SPLINE
SPL {X  -158.264, Y  +691.203, Z    +0.000, E1   -17.264, E3 +51603.968}
SPL {X  -159.000, Y  +685.560, Z    +0.000, E1   -12.398, E3 +51625.143}
SPL {X  -159.924, Y  +672.625, Z    +0.000, E1    -3.689, E3 +51640.160}
SPL {X  -160.000, Y  +663.203, Z    +0.000, E1    +3.155, E3 +51646.815}
SPL {X  -160.000, Y  +652.103, Z    +0.000, E1   +11.247, E3 +51658.485}
SPL {X  -160.000, Y  +641.822, Z    +0.000, E1   +17.059, E3 +51677.859}
SPL {X  -160.000, Y  +631.293, Z    +0.000, E1   +20.354, E3 +51711.738}
SPL {X  -160.000, Y  +627.542, Z    +0.000, E1   +20.380, E3 +51733.145}
SPL {X  -160.000, Y  +623.532, Z    +0.000, E1   +20.378, E3 +51756.111}
SPL {X  -160.000, Y  +619.329, Z    +0.000, E1   +20.391, E3 +51780.148}
SPL {X  -160.000, Y  +614.967, Z    +0.000, E1   +20.392, E3 +51805.128}
SPL {X  -160.000, Y  +611.206, Z    +0.000, E1   +20.351, E3 +51826.800}
SPL {X  -160.000, Y  +607.824, Z    +0.000, E1   +20.354, E3 +51846.221}
SPL {X  -160.000, Y  +603.899, Z    +0.000, E1   +20.373, E3 +51868.671}
SPL {X  -160.000, Y  +599.617, Z    +0.000, E1   +20.384, E3 +51893.164}
SPL {X  -160.000, Y  +595.532, Z    +0.000, E1   +20.373, E3 +51916.525}
SPL {X  -160.000, Y  +591.705, Z    +0.000, E1   +20.373, E3 +51938.450}
SPL {X  -160.000, Y  +588.037, Z    +0.000, E1   +20.359, E3 +51959.537}
SPL {X  -160.000, Y  +584.320, Z    +0.000, E1   +20.364, E3 +51980.838}
SPL {X  -160.000, Y  +580.616, Z    +0.000, E1   +20.357, E3 +52002.065}
SPL {X  -160.000, Y  +577.083, Z    +0.000, E1   +20.358, E3 +52022.314}
SPL {X  -160.000, Y  +573.158, Z    +0.000, E1   +20.377, E3 +52044.766}
SPL {X  -160.000, Y  +568.802, Z    +0.000, E1   +20.385, E3 +52069.718}
SPL {X  -160.000, Y  +564.937, Z    +0.000, E1   +20.350, E3 +52091.938}
SPL {X  -160.000, Y  +561.213, Z    +0.000, E1   +20.372, E3 +52113.225}
SPL {X  -160.000, Y  +557.320, Z    +0.000, E1   +20.363, E3 +52135.551}
SPL {X  -160.000, Y  +553.712, Z    +0.000, E1   +20.355, E3 +52156.251}
SPL {X  -160.000, Y  +550.040, Z    +0.000, E1   +20.360, E3 +52177.289}
SPL {X  -160.000, Y  +546.180, Z    +0.000, E1   +20.370, E3 +52199.345}
SPL {X  -160.000, Y  +542.032, Z    +0.000, E1   +20.384, E3 +52223.084}
SPL {X  -160.000, Y  +537.870, Z    +0.000, E1   +20.372, E3 +52246.959}
SPL {X  -160.000, Y  +534.086, Z    +0.000, E1   +20.356, E3 +52268.713}
SPL {X  -160.000, Y  +530.164, Z    +0.000, E1   +20.382, E3 +52291.063}
SPL {X  -160.000, Y  +527.505, Z    +0.000, E1   +20.318, E3 +52306.436}
SPL {X  -160.000, Y  +511.620, Z    +0.000, E1   +28.365, E3 +52316.899}
SPL {X  -160.000, Y  +507.906, Z    +0.000, E1   +28.152, E3 +52333.295}
SPL {X  -160.000, Y  +506.085, Z    +0.000, E1   +26.146, E3 +52355.754}
SPL {X  -160.000, Y  +504.342, Z    +0.000, E1   +24.109, E3 +52379.269}
SPL {X  -160.000, Y  +503.002, Z    +0.000, E1   +22.325, E3 +52400.275}
SPL {X  -160.000, Y  +500.783, Z    +0.000, E1   +21.421, E3 +52419.864}
SPL {X  -160.000, Y  +497.229, Z    +0.000, E1   +21.403, E3 +52439.172}
SPL {X  -160.000, Y  +493.901, Z    +0.000, E1   +21.409, E3 +52457.191}
SPL {X  -160.000, Y  +490.791, Z    +0.000, E1   +21.400, E3 +52474.064}
SPL {X  -160.000, Y  +487.647, Z    +0.000, E1   +21.401, E3 +52491.110}
SPL {X  -160.000, Y  +484.273, Z    +0.000, E1   +21.408, E3 +52509.390}
SPL {X  -160.000, Y  +481.093, Z    +0.000, E1   +21.389, E3 +52526.699}
SPL {X  -160.000, Y  +478.021, Z    +0.000, E1   +21.401, E3 +52543.306}
SPL {X  -160.000, Y  +474.639, Z    +0.000, E1   +21.410, E3 +52561.597}
SPL {X  -160.000, Y  +471.343, Z    +0.000, E1   +21.399, E3 +52579.499}
SPL {X  -160.000, Y  +468.133, Z    +0.000, E1   +21.402, E3 +52596.891}
SPL {X  -160.000, Y  +464.638, Z    +0.000, E1   +21.421, E3 +52615.740}
SPL {X  -160.000, Y  +461.045, Z    +0.000, E1   +21.424, E3 +52635.154}
SPL {X  -160.000, Y  +457.606, Z    +0.000, E1   +21.413, E3 +52653.864}
SPL {X  -160.000, Y  +454.417, Z    +0.000, E1   +21.401, E3 +52671.172}
SPL {X  -160.000, Y  +451.425, Z    +0.000, E1   +21.404, E3 +52687.394}
SPL {X  -160.000, Y  +448.039, Z    +0.000, E1   +21.417, E3 +52705.687}
SPL {X  -160.000, Y  +444.787, Z    +0.000, E1   +21.414, E3 +52723.242}
SPL {X  -160.000, Y  +441.637, Z    +0.000, E1   +21.431, E3 +52740.220}
SPL {X  -160.000, Y  +438.199, Z    +0.000, E1   +21.432, E3 +52758.824}
SPL {X  -160.000, Y  +434.875, Z    +0.000, E1   +21.424, E3 +52776.864}
SPL {X  -160.000, Y  +431.689, Z    +0.000, E1   +21.423, E3 +52794.112}
SPL {X  -160.000, Y  +428.451, Z    +0.000, E1   +21.430, E3 +52811.592}
SPL {X  -160.000, Y  +425.120, Z    +0.000, E1   +21.430, E3 +52829.656}
SPL {X  -160.000, Y  +421.671, Z    +0.000, E1   +21.430, E3 +52848.340}
SPL {X  -160.000, Y  +418.225, Z    +0.000, E1   +21.425, E3 +52867.021}
SPL {X  -160.000, Y  +414.956, Z    +0.000, E1   +21.424, E3 +52884.702}
SPL {X  -160.000, Y  +411.834, Z    +0.000, E1   +21.420, E3 +52901.620}
SPL {X  -160.000, Y  +408.570, Z    +0.000, E1   +21.432, E3 +52919.229}
SPL {X  -160.000, Y  +405.237, Z    +0.000, E1   +21.432, E3 +52937.258}
SPL {X  -160.000, Y  +402.004, Z    +0.000, E1   +21.424, E3 +52954.833}
SPL {X  -160.000, Y  +398.626, Z    +0.000, E1   +21.425, E3 +52973.139}
SPL {X  -160.000, Y  +395.405, Z    +0.000, E1   +21.422, E3 +52990.557}
SPL {X  -160.000, Y  +392.641, Z    +0.000, E1   +21.407, E3 +53005.555}
SPL {X  -159.989, Y  +390.129, Z    +0.000, E1   +21.406, E3 +53019.196}
SPL {X  -159.932, Y  +387.337, Z    +0.000, E1   +21.403, E3 +53034.392}
SPL {X  -159.823, Y  +384.478, Z    +0.000, E1   +21.379, E3 +53050.055}
SPL {X  -159.660, Y  +381.581, Z    +0.000, E1   +21.363, E3 +53065.943}
SPL {X  -159.452, Y  +378.773, Z    +0.000, E1   +21.330, E3 +53081.390}
SPL {X  -159.222, Y  +376.244, Z    +0.000, E1   +21.297, E3 +53095.352}
SPL {X  -158.814, Y  +372.556, Z    +0.000, E1   +21.316, E3 +53115.619}
SPL {X  -158.301, Y  +368.743, Z    +0.000, E1   +21.199, E3 +53136.941}
SPL {X  -157.981, Y  +366.660, Z    +0.000, E1   +19.986, E3 +53159.909}
ENDSPLINE

SPLINE
SPL {X  -158.491, Y  +370.077, Z    +0.000, E1   +15.910, E3 +53184.922}
SPL {X  -159.771, Y  +383.450, Z    +0.000, E1    +6.314, E3 +53208.077}
SPL {X  -160.000, Y  +392.463, Z    +0.000, E1    +0.112, E3 +53214.584}
SPL {X  -160.000, Y  +399.874, Z    +0.000, E1    -5.508, E3 +53219.086}
SPL {X  -160.000, Y  +411.622, Z    +0.000, E1   -13.815, E3 +53231.206}
SPL {X  -160.000, Y  +419.836, Z    +0.000, E1   -18.198, E3 +53246.380}
SPL {X  -160.000, Y  +430.523, Z    +0.000, E1   -21.710, E3 +53276.580}
SPL {X  -160.000, Y  +433.426, Z    +0.000, E1   -21.735, E3 +53291.994}
SPL {X  -160.000, Y  +436.131, Z    +0.000, E1   -21.710, E3 +53306.469}
SPL {X  -160.000, Y  +439.046, Z    +0.000, E1   -21.732, E3 +53321.963}
SPL {X  -160.000, Y  +442.009, Z    +0.000, E1   -21.719, E3 +53337.785}
SPL {X  -160.000, Y  +444.891, Z    +0.000, E1   -21.724, E3 +53353.140}
SPL {X  -160.000, Y  +449.017, Z    +0.000, E1   -21.792, E3 +53374.932}
SPL {X  -160.000, Y  +452.864, Z    +0.000, E1   -21.730, E3 +53395.550}
SPL {X  -160.000, Y  +455.470, Z    +0.000, E1   -21.722, E3 +53409.439}
SPL {X  -160.000, Y  +458.295, Z    +0.000, E1   -21.738, E3 +53424.460}
SPL {X  -160.000, Y  +461.133, Z    +0.000, E1   -21.720, E3 +53439.642}
SPL {X  -160.000, Y  +464.458, Z    +0.000, E1   -21.770, E3 +53457.161}
SPL {X  -160.000, Y  +468.250, Z    +0.000, E1   -21.764, E3 +53477.314}
SPL {X  -160.000, Y  +472.226, Z    +0.000, E1   -21.782, E3 +53498.473}
SPL {X  -160.000, Y  +476.333, Z    +0.000, E1   -21.767, E3 +53520.387}
SPL {X  -160.000, Y  +480.244, Z    +0.000, E1   -21.765, E3 +53541.252}
SPL {X  -160.000, Y  +484.301, Z    +0.000, E1   -21.775, E3 +53562.780}
SPL {X  -160.000, Y  +488.201, Z    +0.000, E1   -21.768, E3 +53583.540}
SPL {X  -160.000, Y  +492.394, Z    +0.000, E1   -21.802, E3 +53605.714}
SPL {X  -160.000, Y  +496.781, Z    +0.000, E1   -21.798, E3 +53629.026}
SPL {X  -160.000, Y  +501.083, Z    +0.000, E1   -21.796, E3 +53651.956}
SPL {X  -160.000, Y  +504.917, Z    +0.000, E1   -21.764, E3 +53672.460}
SPL {X  -160.000, Y  +508.886, Z    +0.000, E1   -21.791, E3 +53693.546}
SPL {X  -160.000, Y  +513.057, Z    +0.000, E1   -21.767, E3 +53715.854}
SPL {X  -160.000, Y  +517.221, Z    +0.000, E1   -21.778, E3 +53738.006}
SPL {X  -160.000, Y  +521.677, Z    +0.000, E1   -21.781, E3 +53761.768}
SPL {X  -160.000, Y  +525.729, Z    +0.000, E1   -21.753, E3 +53783.407}
SPL {X  -160.000, Y  +529.456, Z    +0.000, E1   -21.766, E3 +53803.186}
SPL {X  -160.000, Y  +533.608, Z    +0.000, E1   -21.776, E3 +53825.317}
SPL {X  -160.000, Y  +538.227, Z    +0.000, E1   -21.794, E3 +53849.849}
SPL {X  -160.000, Y  +542.483, Z    +0.000, E1   -21.764, E3 +53872.574}
SPL {X  -160.000, Y  +546.194, Z    +0.000, E1   -21.754, E3 +53892.391}
SPL {X  -160.000, Y  +550.131, Z    +0.000, E1   -21.771, E3 +53913.327}
SPL {X  -160.000, Y  +554.462, Z    +0.000, E1   -21.777, E3 +53936.381}
SPL {X  -160.000, Y  +558.542, Z    +0.000, E1   -21.758, E3 +53958.153}
SPL {X  -160.000, Y  +562.615, Z    +0.000, E1   -21.776, E3 +53979.809}
SPL {X  -160.000, Y  +566.764, Z    +0.000, E1   -21.764, E3 +54001.934}
SPL {X  -160.000, Y  +570.657, Z    +0.000, E1   -21.758, E3 +54022.681}
SPL {X  -160.000, Y  +574.688, Z    +0.000, E1   -21.771, E3 +54044.124}
SPL {X  -160.000, Y  +578.864, Z    +0.000, E1   -21.770, E3 +54066.375}
SPL {X  -160.000, Y  +582.807, Z    +0.000, E1   -21.754, E3 +54087.429}
SPL {X  -160.000, Y  +586.993, Z    +0.000, E1   -21.779, E3 +54109.665}
SPL {X  -160.000, Y  +591.368, Z    +0.000, E1   -21.775, E3 +54132.952}
SPL {X  -160.000, Y  +595.703, Z    +0.000, E1   -21.775, E3 +54156.061}
SPL {X  -160.000, Y  +599.558, Z    +0.000, E1   -21.748, E3 +54176.639}
SPL {X  -160.000, Y  +603.126, Z    +0.000, E1   -21.757, E3 +54195.618}
SPL {X  -160.000, Y  +607.107, Z    +0.000, E1   -21.766, E3 +54216.843}
SPL {X  -160.000, Y  +611.246, Z    +0.000, E1   -21.760, E3 +54238.917}
SPL {X  -160.000, Y  +615.151, Z    +0.000, E1   -21.752, E3 +54259.730}
SPL {X  -160.000, Y  +618.728, Z    +0.000, E1   -21.747, E3 +54278.792}
SPL {X  -160.000, Y  +622.318, Z    +0.000, E1   -21.753, E3 +54297.907}
SPL {X  -160.000, Y  +625.877, Z    +0.000, E1   -21.745, E3 +54316.885}
SPL {X  -160.000, Y  +629.892, Z    +0.000, E1   -21.777, E3 +54338.209}
SPL {X  -160.000, Y  +634.024, Z    +0.000, E1   -21.756, E3 +54360.259}
SPL {X  -160.000, Y  +637.661, Z    +0.000, E1   -21.748, E3 +54379.650}
SPL {X  -160.000, Y  +641.244, Z    +0.000, E1   -21.752, E3 +54398.721}
SPL {X  -160.000, Y  +645.120, Z    +0.000, E1   -21.762, E3 +54419.353}
SPL {X  -160.000, Y  +649.214, Z    +0.000, E1   -21.766, E3 +54441.141}
SPL {X  -160.000, Y  +653.188, Z    +0.000, E1   -21.771, E3 +54462.204}
SPL {X  -160.000, Y  +656.905, Z    +0.000, E1   -21.769, E3 +54481.979}
SPL {X  -160.000, Y  +660.685, Z    +0.000, E1   -21.769, E3 +54502.147}
SPL {X  -160.000, Y  +664.985, Z    +0.000, E1   -21.790, E3 +54525.000}
SPL {X  -159.993, Y  +669.170, Z    +0.000, E1   -21.763, E3 +54547.358}
SPL {X  -159.916, Y  +672.869, Z    +0.000, E1   -21.755, E3 +54567.103}
SPL {X  -159.752, Y  +676.610, Z    +0.000, E1   -21.740, E3 +54587.178}
SPL {X  -159.478, Y  +680.618, Z    +0.000, E1   -21.719, E3 +54608.777}
SPL {X  -159.108, Y  +684.576, Z    +0.000, E1   -21.664, E3 +54630.247}
SPL {X  -158.638, Y  +688.530, Z    +0.000, E1   -21.617, E3 +54651.768}
SPL {X  -158.097, Y  +692.303, Z    +0.000, E1   -21.529, E3 +54672.486}
ENDSPLINE

SPLINE
SPL {X  -158.264, Y  +691.203, Z    +0.000, E1   -17.264, E3 +54709.231}
SPL {X  -159.000, Y  +685.560, Z    +0.000, E1   -12.398, E3 +54730.407}
SPL {X  -159.924, Y  +672.625, Z    +0.000, E1    -3.689, E3 +54745.424}
SPL {X  -160.000, Y  +663.203, Z    +0.000, E1    +3.155, E3 +54752.078}
SPL {X  -160.000, Y  +652.103, Z    +0.000, E1   +11.247, E3 +54763.748}
SPL {X  -160.000, Y  +641.822, Z    +0.000, E1   +17.059, E3 +54783.122}
SPL {X  -160.000, Y  +631.293, Z    +0.000, E1   +20.354, E3 +54817.002}
SPL {X  -160.000, Y  +627.542, Z    +0.000, E1   +20.380, E3 +54838.409}
SPL {X  -160.000, Y  +623.532, Z    +0.000, E1   +20.378, E3 +54861.374}
SPL {X  -160.000, Y  +619.329, Z    +0.000, E1   +20.391, E3 +54885.412}
SPL {X  -160.000, Y  +614.967, Z    +0.000, E1   +20.392, E3 +54910.392}
SPL {X  -160.000, Y  +611.206, Z    +0.000, E1   +20.351, E3 +54932.063}
SPL {X  -160.000, Y  +607.824, Z    +0.000, E1   +20.354, E3 +54951.484}
SPL {X  -160.000, Y  +603.899, Z    +0.000, E1   +20.373, E3 +54973.934}
SPL {X  -160.000, Y  +599.617, Z    +0.000, E1   +20.384, E3 +54998.428}
SPL {X  -160.000, Y  +595.532, Z    +0.000, E1   +20.373, E3 +55021.788}
SPL {X  -160.000, Y  +591.705, Z    +0.000, E1   +20.373, E3 +55043.713}
SPL {X  -160.000, Y  +588.037, Z    +0.000, E1   +20.359, E3 +55064.800}
SPL {X  -160.000, Y  +584.320, Z    +0.000, E1   +20.364, E3 +55086.102}
SPL {X  -160.000, Y  +580.616, Z    +0.000, E1   +20.357, E3 +55107.329}
SPL {X  -160.000, Y  +577.083, Z    +0.000, E1   +20.358, E3 +55127.577}
SPL {X  -160.000, Y  +573.158, Z    +0.000, E1   +20.377, E3 +55150.029}
SPL {X  -160.000, Y  +568.802, Z    +0.000, E1   +20.385, E3 +55174.981}
SPL {X  -160.000, Y  +564.937, Z    +0.000, E1   +20.350, E3 +55197.202}
SPL {X  -160.000, Y  +561.213, Z    +0.000, E1   +20.372, E3 +55218.488}
SPL {X  -160.000, Y  +557.320, Z    +0.000, E1   +20.363, E3 +55240.815}
SPL {X  -160.000, Y  +553.712, Z    +0.000, E1   +20.355, E3 +55261.514}
SPL {X  -160.000, Y  +550.040, Z    +0.000, E1   +20.360, E3 +55282.552}
SPL {X  -160.000, Y  +546.180, Z    +0.000, E1   +20.370, E3 +55304.608}
SPL {X  -160.000, Y  +542.032, Z    +0.000, E1   +20.384, E3 +55328.347}
SPL {X  -160.000, Y  +537.870, Z    +0.000, E1   +20.372, E3 +55352.223}
SPL {X  -160.000, Y  +534.086, Z    +0.000, E1   +20.356, E3 +55373.977}
SPL {X  -160.000, Y  +530.164, Z    +0.000, E1   +20.382, E3 +55396.326}
SPL {X  -160.000, Y  +527.505, Z    +0.000, E1   +20.318, E3 +55411.700}
SPL {X  -160.000, Y  +511.620, Z    +0.000, E1   +28.365, E3 +55422.163}
SPL {X  -160.000, Y  +507.906, Z    +0.000, E1   +28.152, E3 +55438.558}
SPL {X  -160.000, Y  +506.085, Z    +0.000, E1   +26.146, E3 +55461.018}
SPL {X  -160.000, Y  +504.342, Z    +0.000, E1   +24.109, E3 +55484.533}
SPL {X  -160.000, Y  +503.002, Z    +0.000, E1   +22.325, E3 +55505.538}
SPL {X  -160.000, Y  +500.783, Z    +0.000, E1   +21.421, E3 +55525.127}
SPL {X  -160.000, Y  +497.229, Z    +0.000, E1   +21.403, E3 +55544.435}
SPL {X  -160.000, Y  +493.901, Z    +0.000, E1   +21.409, E3 +55562.454}
SPL {X  -160.000, Y  +490.791, Z    +0.000, E1   +21.400, E3 +55579.327}
SPL {X  -160.000, Y  +487.647, Z    +0.000, E1   +21.401, E3 +55596.374}
SPL {X  -160.000, Y  +484.273, Z    +0.000, E1   +21.408, E3 +55614.654}
SPL {X  -160.000, Y  +481.093, Z    +0.000, E1   +21.389, E3 +55631.963}
SPL {X  -160.000, Y  +478.021, Z    +0.000, E1   +21.401, E3 +55648.569}
SPL {X  -160.000, Y  +474.639, Z    +0.000, E1   +21.410, E3 +55666.861}
SPL {X  -160.000, Y  +471.343, Z    +0.000, E1   +21.399, E3 +55684.763}
SPL {X  -160.000, Y  +468.133, Z    +0.000, E1   +21.402, E3 +55702.154}
SPL {X  -160.000, Y  +464.638, Z    +0.000, E1   +21.421, E3 +55721.003}
SPL {X  -160.000, Y  +461.045, Z    +0.000, E1   +21.424, E3 +55740.417}
SPL {X  -160.000, Y  +457.606, Z    +0.000, E1   +21.413, E3 +55759.127}
SPL {X  -160.000, Y  +454.417, Z    +0.000, E1   +21.401, E3 +55776.436}
SPL {X  -160.000, Y  +451.425, Z    +0.000, E1   +21.404, E3 +55792.657}
SPL {X  -160.000, Y  +448.039, Z    +0.000, E1   +21.417, E3 +55810.950}
SPL {X  -160.000, Y  +444.787, Z    +0.000, E1   +21.414, E3 +55828.505}
SPL {X  -160.000, Y  +441.637, Z    +0.000, E1   +21.431, E3 +55845.483}
SPL {X  -160.000, Y  +438.199, Z    +0.000, E1   +21.432, E3 +55864.087}
SPL {X  -160.000, Y  +434.875, Z    +0.000, E1   +21.424, E3 +55882.127}
SPL {X  -160.000, Y  +431.689, Z    +0.000, E1   +21.423, E3 +55899.375}
SPL {X  -160.000, Y  +428.451, Z    +0.000, E1   +21.430, E3 +55916.855}
SPL {X  -160.000, Y  +425.120, Z    +0.000, E1   +21.430, E3 +55934.919}
SPL {X  -160.000, Y  +421.671, Z    +0.000, E1   +21.430, E3 +55953.603}
SPL {X  -160.000, Y  +418.225, Z    +0.000, E1   +21.425, E3 +55972.285}
SPL {X  -160.000, Y  +414.956, Z    +0.000, E1   +21.424, E3 +55989.966}
SPL {X  -160.000, Y  +411.834, Z    +0.000, E1   +21.420, E3 +56006.884}
SPL {X  -160.000, Y  +408.570, Z    +0.000, E1   +21.432, E3 +56024.493}
SPL {X  -160.000, Y  +405.237, Z    +0.000, E1   +21.432, E3 +56042.521}
SPL {X  -160.000, Y  +402.004, Z    +0.000, E1   +21.424, E3 +56060.097}
SPL {X  -160.000, Y  +398.626, Z    +0.000, E1   +21.425, E3 +56078.403}
SPL {X  -160.000, Y  +395.405, Z    +0.000, E1   +21.422, E3 +56095.820}
SPL {X  -160.000, Y  +392.641, Z    +0.000, E1   +21.407, E3 +56110.819}
SPL {X  -159.989, Y  +390.129, Z    +0.000, E1   +21.406, E3 +56124.459}
SPL {X  -159.932, Y  +387.337, Z    +0.000, E1   +21.403, E3 +56139.655}
SPL {X  -159.823, Y  +384.478, Z    +0.000, E1   +21.379, E3 +56155.318}
SPL {X  -159.660, Y  +381.581, Z    +0.000, E1   +21.363, E3 +56171.207}
SPL {X  -159.452, Y  +378.773, Z    +0.000, E1   +21.330, E3 +56186.653}
SPL {X  -159.222, Y  +376.244, Z    +0.000, E1   +21.297, E3 +56200.615}
SPL {X  -158.814, Y  +372.556, Z    +0.000, E1   +21.316, E3 +56220.883}
SPL {X  -158.301, Y  +368.743, Z    +0.000, E1   +21.199, E3 +56242.205}
SPL {X  -157.981, Y  +366.660, Z    +0.000, E1   +19.986, E3 +56265.172}
ENDSPLINE

SPLINE
SPL {X  -158.491, Y  +370.077, Z    +0.000, E1   +15.910, E3 +56290.185}
SPL {X  -159.771, Y  +383.450, Z    +0.000, E1    +6.314, E3 +56313.340}
SPL {X  -160.000, Y  +392.463, Z    +0.000, E1    +0.112, E3 +56319.847}
SPL {X  -160.000, Y  +399.874, Z    +0.000, E1    -5.508, E3 +56324.350}
SPL {X  -160.000, Y  +411.622, Z    +0.000, E1   -13.815, E3 +56336.470}
SPL {X  -160.000, Y  +419.836, Z    +0.000, E1   -18.198, E3 +56351.643}
SPL {X  -160.000, Y  +430.523, Z    +0.000, E1   -21.710, E3 +56381.843}
SPL {X  -160.000, Y  +433.426, Z    +0.000, E1   -21.735, E3 +56397.258}
SPL {X  -160.000, Y  +436.131, Z    +0.000, E1   -21.710, E3 +56411.733}
SPL {X  -160.000, Y  +439.046, Z    +0.000, E1   -21.732, E3 +56427.226}
SPL {X  -160.000, Y  +442.009, Z    +0.000, E1   -21.719, E3 +56443.048}
SPL {X  -160.000, Y  +444.891, Z    +0.000, E1   -21.724, E3 +56458.404}
SPL {X  -160.000, Y  +449.017, Z    +0.000, E1   -21.792, E3 +56480.196}
SPL {X  -160.000, Y  +452.864, Z    +0.000, E1   -21.730, E3 +56500.813}
SPL {X  -160.000, Y  +455.470, Z    +0.000, E1   -21.722, E3 +56514.702}
SPL {X  -160.000, Y  +458.295, Z    +0.000, E1   -21.738, E3 +56529.723}
SPL {X  -160.000, Y  +461.133, Z    +0.000, E1   -21.720, E3 +56544.906}
SPL {X  -160.000, Y  +464.458, Z    +0.000, E1   -21.770, E3 +56562.425}
SPL {X  -160.000, Y  +468.250, Z    +0.000, E1   -21.764, E3 +56582.578}
SPL {X  -160.000, Y  +472.226, Z    +0.000, E1   -21.782, E3 +56603.736}
SPL {X  -160.000, Y  +476.333, Z    +0.000, E1   -21.767, E3 +56625.651}
SPL {X  -160.000, Y  +480.244, Z    +0.000, E1   -21.765, E3 +56646.515}
SPL {X  -160.000, Y  +484.301, Z    +0.000, E1   -21.775, E3 +56668.044}
SPL {X  -160.000, Y  +488.201, Z    +0.000, E1   -21.768, E3 +56688.803}
SPL {X  -160.000, Y  +492.394, Z    +0.000, E1   -21.802, E3 +56710.978}
SPL {X  -160.000, Y  +496.781, Z    +0.000, E1   -21.798, E3 +56734.289}
SPL {X  -160.000, Y  +501.083, Z    +0.000, E1   -21.796, E3 +56757.219}
SPL {X  -160.000, Y  +504.917, Z    +0.000, E1   -21.764, E3 +56777.724}
SPL {X  -160.000, Y  +508.886, Z    +0.000, E1   -21.791, E3 +56798.810}
SPL {X  -160.000, Y  +513.057, Z    +0.000, E1   -21.767, E3 +56821.117}
SPL {X  -160.000, Y  +517.221, Z    +0.000, E1   -21.778, E3 +56843.270}
SPL {X  -160.000, Y  +521.677, Z    +0.000, E1   -21.781, E3 +56867.031}
SPL {X  -160.000, Y  +525.729, Z    +0.000, E1   -21.753, E3 +56888.671}
SPL {X  -160.000, Y  +529.456, Z    +0.000, E1   -21.766, E3 +56908.450}
SPL {X  -160.000, Y  +533.608, Z    +0.000, E1   -21.776, E3 +56930.580}
SPL {X  -160.000, Y  +538.227, Z    +0.000, E1   -21.794, E3 +56955.113}
SPL {X  -160.000, Y  +542.483, Z    +0.000, E1   -21.764, E3 +56977.838}
SPL {X  -160.000, Y  +546.194, Z    +0.000, E1   -21.754, E3 +56997.654}
SPL {X  -160.000, Y  +550.131, Z    +0.000, E1   -21.771, E3 +57018.590}
SPL {X  -160.000, Y  +554.462, Z    +0.000, E1   -21.777, E3 +57041.644}
SPL {X  -160.000, Y  +558.542, Z    +0.000, E1   -21.758, E3 +57063.417}
SPL {X  -160.000, Y  +562.615, Z    +0.000, E1   -21.776, E3 +57085.073}
SPL {X  -160.000, Y  +566.764, Z    +0.000, E1   -21.764, E3 +57107.197}
SPL {X  -160.000, Y  +570.657, Z    +0.000, E1   -21.758, E3 +57127.945}
SPL {X  -160.000, Y  +574.688, Z    +0.000, E1   -21.771, E3 +57149.388}
SPL {X  -160.000, Y  +578.864, Z    +0.000, E1   -21.770, E3 +57171.638}
SPL {X  -160.000, Y  +582.807, Z    +0.000, E1   -21.754, E3 +57192.693}
SPL {X  -160.000, Y  +586.993, Z    +0.000, E1   -21.779, E3 +57214.928}
SPL {X  -160.000, Y  +591.368, Z    +0.000, E1   -21.775, E3 +57238.215}
SPL {X  -160.000, Y  +595.703, Z    +0.000, E1   -21.775, E3 +57261.325}
SPL {X  -160.000, Y  +599.558, Z    +0.000, E1   -21.748, E3 +57281.902}
SPL {X  -160.000, Y  +603.126, Z    +0.000, E1   -21.757, E3 +57300.882}
SPL {X  -160.000, Y  +607.107, Z    +0.000, E1   -21.766, E3 +57322.107}
SPL {X  -160.000, Y  +611.246, Z    +0.000, E1   -21.760, E3 +57344.180}
SPL {X  -160.000, Y  +615.151, Z    +0.000, E1   -21.752, E3 +57364.993}
SPL {X  -160.000, Y  +618.728, Z    +0.000, E1   -21.747, E3 +57384.056}
SPL {X  -160.000, Y  +622.318, Z    +0.000, E1   -21.753, E3 +57403.170}
SPL {X  -160.000, Y  +625.877, Z    +0.000, E1   -21.745, E3 +57422.149}
SPL {X  -160.000, Y  +629.892, Z    +0.000, E1   -21.777, E3 +57443.472}
SPL {X  -160.000, Y  +634.024, Z    +0.000, E1   -21.756, E3 +57465.523}
SPL {X  -160.000, Y  +637.661, Z    +0.000, E1   -21.748, E3 +57484.913}
SPL {X  -160.000, Y  +641.244, Z    +0.000, E1   -21.752, E3 +57503.984}
SPL {X  -160.000, Y  +645.120, Z    +0.000, E1   -21.762, E3 +57524.616}
SPL {X  -160.000, Y  +649.214, Z    +0.000, E1   -21.766, E3 +57546.405}
SPL {X  -160.000, Y  +653.188, Z    +0.000, E1   -21.771, E3 +57567.467}
SPL {X  -160.000, Y  +656.905, Z    +0.000, E1   -21.769, E3 +57587.243}
SPL {X  -160.000, Y  +660.685, Z    +0.000, E1   -21.769, E3 +57607.410}
SPL {X  -160.000, Y  +664.985, Z    +0.000, E1   -21.790, E3 +57630.263}
SPL {X  -159.993, Y  +669.170, Z    +0.000, E1   -21.763, E3 +57652.622}
SPL {X  -159.916, Y  +672.869, Z    +0.000, E1   -21.755, E3 +57672.367}
SPL {X  -159.752, Y  +676.610, Z    +0.000, E1   -21.740, E3 +57692.441}
SPL {X  -159.478, Y  +680.618, Z    +0.000, E1   -21.719, E3 +57714.041}
SPL {X  -159.108, Y  +684.576, Z    +0.000, E1   -21.664, E3 +57735.510}
SPL {X  -158.638, Y  +688.530, Z    +0.000, E1   -21.617, E3 +57757.032}
SPL {X  -158.097, Y  +692.303, Z    +0.000, E1   -21.529, E3 +57777.749}
ENDSPLINE

SPLINE
SPL {X  -158.264, Y  +691.203, Z    +0.000, E1   -17.264, E3 +57814.495}
SPL {X  -159.000, Y  +685.560, Z    +0.000, E1   -12.398, E3 +57835.670}
SPL {X  -159.924, Y  +672.625, Z    +0.000, E1    -3.689, E3 +57850.687}
SPL {X  -160.000, Y  +663.203, Z    +0.000, E1    +3.155, E3 +57857.342}
SPL {X  -160.000, Y  +652.103, Z    +0.000, E1   +11.247, E3 +57869.012}
SPL {X  -160.000, Y  +641.822, Z    +0.000, E1   +17.059, E3 +57888.386}
SPL {X  -160.000, Y  +631.293, Z    +0.000, E1   +20.354, E3 +57922.265}
SPL {X  -160.000, Y  +627.542, Z    +0.000, E1   +20.380, E3 +57943.672}
SPL {X  -160.000, Y  +623.532, Z    +0.000, E1   +20.378, E3 +57966.638}
SPL {X  -160.000, Y  +619.329, Z    +0.000, E1   +20.391, E3 +57990.675}
SPL {X  -160.000, Y  +614.967, Z    +0.000, E1   +20.392, E3 +58015.655}
SPL {X  -160.000, Y  +611.206, Z    +0.000, E1   +20.351, E3 +58037.327}
SPL {X  -160.000, Y  +607.824, Z    +0.000, E1   +20.354, E3 +58056.748}
SPL {X  -160.000, Y  +603.899, Z    +0.000, E1   +20.373, E3 +58079.198}
SPL {X  -160.000, Y  +599.617, Z    +0.000, E1   +20.384, E3 +58103.692}
SPL {X  -160.000, Y  +595.532, Z    +0.000, E1   +20.373, E3 +58127.052}
SPL {X  -160.000, Y  +591.705, Z    +0.000, E1   +20.373, E3 +58148.977}
SPL {X  -160.000, Y  +588.037, Z    +0.000, E1   +20.359, E3 +58170.064}
SPL {X  -160.000, Y  +584.320, Z    +0.000, E1   +20.364, E3 +58191.365}
SPL {X  -160.000, Y  +580.616, Z    +0.000, E1   +20.357, E3 +58212.592}
SPL {X  -160.000, Y  +577.083, Z    +0.000, E1   +20.358, E3 +58232.841}
SPL {X  -160.000, Y  +573.158, Z    +0.000, E1   +20.377, E3 +58255.293}
SPL {X  -160.000, Y  +568.802, Z    +0.000, E1   +20.385, E3 +58280.245}
SPL {X  -160.000, Y  +564.937, Z    +0.000, E1   +20.350, E3 +58302.465}
SPL {X  -160.000, Y  +561.213, Z    +0.000, E1   +20.372, E3 +58323.752}
SPL {X  -160.000, Y  +557.320, Z    +0.000, E1   +20.363, E3 +58346.078}
SPL {X  -160.000, Y  +553.712, Z    +0.000, E1   +20.355, E3 +58366.778}
SPL {X  -160.000, Y  +550.040, Z    +0.000, E1   +20.360, E3 +58387.816}
SPL {X  -160.000, Y  +546.180, Z    +0.000, E1   +20.370, E3 +58409.872}
SPL {X  -160.000, Y  +542.032, Z    +0.000, E1   +20.384, E3 +58433.611}
SPL {X  -160.000, Y  +537.870, Z    +0.000, E1   +20.372, E3 +58457.486}
SPL {X  -160.000, Y  +534.086, Z    +0.000, E1   +20.356, E3 +58479.240}
SPL {X  -160.000, Y  +530.164, Z    +0.000, E1   +20.382, E3 +58501.590}
SPL {X  -160.000, Y  +527.505, Z    +0.000, E1   +20.318, E3 +58516.963}
SPL {X  -160.000, Y  +511.620, Z    +0.000, E1   +28.365, E3 +58527.426}
SPL {X  -160.000, Y  +507.906, Z    +0.000, E1   +28.152, E3 +58543.822}
SPL {X  -160.000, Y  +506.085, Z    +0.000, E1   +26.146, E3 +58566.281}
SPL {X  -160.000, Y  +504.342, Z    +0.000, E1   +24.109, E3 +58589.796}
SPL {X  -160.000, Y  +503.002, Z    +0.000, E1   +22.325, E3 +58610.802}
ENDSPLINE

SPLINE
SPL {X  -160.000, Y  +512.244, Z    +0.000, E1   +14.473, E3 +58629.538}
SPL {X  -160.000, Y  +509.675, Z    +0.000, E1   +14.481, E3 +58650.682}
SPL {X  -160.000, Y  +507.162, Z    +0.000, E1   +14.470, E3 +58671.422}
SPL {X  -160.000, Y  +504.735, Z    +0.000, E1   +14.473, E3 +58691.393}
SPL {X  -160.000, Y  +502.261, Z    +0.000, E1   +14.476, E3 +58711.729}
SPL {X  -160.000, Y  +499.798, Z    +0.000, E1   +14.482, E3 +58731.932}
SPL {X  -160.000, Y  +497.435, Z    +0.000, E1   +14.476, E3 +58751.408}
SPL {X  -160.000, Y  +495.089, Z    +0.000, E1   +14.475, E3 +58770.775}
SPL {X  -160.000, Y  +492.764, Z    +0.000, E1   +14.469, E3 +58789.947}
SPL {X  -160.000, Y  +490.292, Z    +0.000, E1   +14.476, E3 +58810.348}
SPL {X  -160.000, Y  +487.641, Z    +0.000, E1   +14.470, E3 +58832.244}
SPL {X  -160.000, Y  +485.054, Z    +0.000, E1   +14.460, E3 +58853.686}
SPL {X  -160.000, Y  +482.421, Z    +0.000, E1   +14.461, E3 +58875.405}
SPL {X  -160.000, Y  +480.000, Z    +0.000, E1   +14.451, E3 +58895.369}
SPL {X  -160.000, Y  +477.551, Z    +0.000, E1   +14.466, E3 +58915.497}
SPL {X  -160.000, Y  +475.253, Z    +0.000, E1   +14.450, E3 +58934.471}
SPL {X  -160.000, Y  +473.070, Z    +0.000, E1   +14.454, E3 +58952.492}
SPL {X  -160.000, Y  +470.603, Z    +0.000, E1   +14.464, E3 +58972.793}
SPL {X  -160.000, Y  +468.243, Z    +0.000, E1   +14.458, E3 +58992.192}
SPL {X  -160.000, Y  +465.791, Z    +0.000, E1   +14.475, E3 +59012.336}
SPL {X  -160.000, Y  +463.103, Z    +0.000, E1   +14.474, E3 +59034.485}
SPL {X  -160.000, Y  +460.743, Z    +0.000, E1   +14.465, E3 +59053.893}
SPL {X  -160.000, Y  +458.292, Z    +0.000, E1   +14.492, E3 +59073.892}
SPL {X  -160.000, Y  +455.874, Z    +0.000, E1   +14.484, E3 +59093.750}
SPL {X  -160.000, Y  +453.555, Z    +0.000, E1   +14.488, E3 +59112.829}
SPL {X  -160.000, Y  +451.093, Z    +0.000, E1   +14.485, E3 +59133.141}
SPL {X  -160.000, Y  +448.700, Z    +0.000, E1   +14.483, E3 +59152.831}
SPL {X  -160.000, Y  +446.277, Z    +0.000, E1   +14.485, E3 +59172.754}
SPL {X  -160.000, Y  +443.879, Z    +0.000, E1   +14.485, E3 +59192.492}
SPL {X  -160.000, Y  +441.447, Z    +0.000, E1   +14.485, E3 +59212.500}
SPL {X  -160.000, Y  +439.006, Z    +0.000, E1   +14.488, E3 +59232.583}
SPL {X  -160.000, Y  +436.311, Z    +0.000, E1   +14.498, E3 +59254.742}
SPL {X  -160.000, Y  +433.559, Z    +0.000, E1   +14.491, E3 +59277.411}
SPL {X  -160.000, Y  +431.162, Z    +0.000, E1   +14.479, E3 +59297.162}
SPL {X  -160.000, Y  +429.152, Z    +0.000, E1   +14.469, E3 +59313.744}
SPL {X  -160.000, Y  +426.863, Z    +0.000, E1   +14.490, E3 +59332.523}
SPL {X  -160.000, Y  +424.653, Z    +0.000, E1   +14.467, E3 +59350.782}
SPL {X  -160.000, Y  +422.337, Z    +0.000, E1   +14.492, E3 +59369.766}
SPL {X  -160.000, Y  +419.639, Z    +0.000, E1   +14.504, E3 +59391.806}
SPL {X  -160.000, Y  +417.127, Z    +0.000, E1   +14.501, E3 +59412.397}
SPL {X  -160.000, Y  +414.849, Z    +0.000, E1   +14.496, E3 +59431.131}
SPL {X  -160.000, Y  +412.396, Z    +0.000, E1   +14.505, E3 +59451.320}
SPL {X  -160.000, Y  +409.815, Z    +0.000, E1   +14.498, E3 +59472.575}
SPL {X  -160.000, Y  +407.614, Z    +0.000, E1   +14.484, E3 +59490.700}
SPL {X  -160.000, Y  +405.406, Z    +0.000, E1   +14.501, E3 +59508.763}
SPL {X  -160.000, Y  +402.958, Z    +0.000, E1   +14.500, E3 +59528.933}
SPL {X  -160.000, Y  +400.690, Z    +0.000, E1   +14.484, E3 +59547.645}
SPL {X  -160.000, Y  +398.391, Z    +0.000, E1   +14.502, E3 +59566.471}
SPL {X  -160.000, Y  +395.999, Z    +0.000, E1   +14.484, E3 +59586.261}
SPL {X  -160.000, Y  +393.685, Z    +0.000, E1   +14.486, E3 +59605.333}
SPL {X  -159.999, Y  +391.313, Z    +0.000, E1   +14.479, E3 +59624.915}
SPL {X  -159.970, Y  +388.900, Z    +0.000, E1   +14.480, E3 +59644.799}
SPL {X  -159.903, Y  +386.417, Z    +0.000, E1   +14.475, E3 +59665.304}
SPL {X  -159.796, Y  +383.921, Z    +0.000, E1   +14.466, E3 +59685.960}
SPL {X  -159.651, Y  +381.443, Z    +0.000, E1   +14.453, E3 +59706.507}
SPL {X  -159.474, Y  +379.042, Z    +0.000, E1   +14.434, E3 +59726.471}
SPL {X  -159.316, Y  +377.219, Z    +0.000, E1   +14.400, E3 +59741.700}
ENDSPLINE

SPLINE
SPL {X  -159.452, Y  +378.767, Z    +0.000, E1   +11.887, E3 +59762.689}
SPL {X  -159.840, Y  +384.856, Z    +0.000, E1    +7.126, E3 +59781.661}
SPL {X  -159.991, Y  +390.336, Z    +0.000, E1    +2.803, E3 +59795.483}
SPL {X  -160.000, Y  +403.532, Z    +0.000, E1    -6.523, E3 +59813.204}
SPL {X  -160.000, Y  +409.023, Z    +0.000, E1   -10.003, E3 +59823.978}
SPL {X  -160.000, Y  +418.032, Z    +0.000, E1   -14.569, E3 +59848.837}
SPL {X  -160.000, Y  +420.561, Z    +0.000, E1   -14.816, E3 +59866.317}
SPL {X  -160.000, Y  +422.801, Z    +0.000, E1   -14.823, E3 +59884.265}
SPL {X  -160.000, Y  +425.518, Z    +0.000, E1   -14.845, E3 +59906.040}
SPL {X  -160.000, Y  +428.688, Z    +0.000, E1   -14.854, E3 +59931.448}
SPL {X  -160.000, Y  +431.971, Z    +0.000, E1   -14.849, E3 +59957.917}
SPL {X  -160.000, Y  +435.345, Z    +0.000, E1   -14.857, E3 +59984.967}
SPL {X  -160.000, Y  +438.732, Z    +0.000, E1   -14.858, E3 +60012.115}
SPL {X  -160.000, Y  +441.925, Z    +0.000, E1   -14.848, E3 +60037.786}
SPL {X  -160.000, Y  +444.299, Z    +0.000, E1   -14.809, E3 +60056.970}
SPL {X  -160.000, Y  +446.229, Z    +0.000, E1   -14.820, E3 +60072.389}
SPL {X  -160.000, Y  +448.987, Z    +0.000, E1   -14.868, E3 +60094.326}
SPL {X  -160.000, Y  +452.351, Z    +0.000, E1   -14.871, E3 +60121.302}
SPL {X  -160.000, Y  +455.709, Z    +0.000, E1   -14.880, E3 +60148.116}
SPL {X  -160.000, Y  +458.189, Z    +0.000, E1   -14.832, E3 +60168.118}
SPL {X  -160.000, Y  +459.885, Z    +0.000, E1   -14.825, E3 +60181.789}
SPL {X  -160.000, Y  +462.438, Z    +0.000, E1   -14.868, E3 +60202.199}
SPL {X  -160.000, Y  +465.575, Z    +0.000, E1   -14.849, E3 +60227.507}
SPL {X  -160.000, Y  +468.581, Z    +0.000, E1   -14.841, E3 +60251.739}
SPL {X  -160.000, Y  +471.795, Z    +0.000, E1   -14.854, E3 +60277.527}
SPL {X  -160.000, Y  +475.138, Z    +0.000, E1   -14.853, E3 +60304.377}
SPL {X  -160.000, Y  +477.981, Z    +0.000, E1   -14.823, E3 +60327.297}
SPL {X  -160.000, Y  +480.658, Z    +0.000, E1   -14.835, E3 +60348.773}
SPL {X  -160.000, Y  +483.534, Z    +0.000, E1   -14.838, E3 +60371.868}
SPL {X  -160.000, Y  +486.226, Z    +0.000, E1   -14.823, E3 +60393.533}
SPL {X  -160.000, Y  +488.751, Z    +0.000, E1   -14.827, E3 +60413.806}
SPL {X  -160.000, Y  +491.612, Z    +0.000, E1   -14.844, E3 +60436.728}
SPL {X  -160.000, Y  +494.417, Z    +0.000, E1   -14.827, E3 +60459.319}
SPL {X  -160.000, Y  +496.961, Z    +0.000, E1   -14.824, E3 +60479.763}
SPL {X  -160.000, Y  +499.610, Z    +0.000, E1   -14.830, E3 +60501.036}
SPL {X  -160.000, Y  +502.268, Z    +0.000, E1   -14.832, E3 +60522.305}
SPL {X  -160.000, Y  +505.041, Z    +0.000, E1   -14.849, E3 +60544.467}
SPL {X  -160.000, Y  +507.743, Z    +0.000, E1   -14.842, E3 +60566.091}
SPL {X  -160.000, Y  +510.437, Z    +0.000, E1   -14.860, E3 +60587.605}
SPL {X  -160.000, Y  +513.179, Z    +0.000, E1   -14.849, E3 +60609.653}
SPL {X  -160.000, Y  +515.613, Z    +0.000, E1   -14.829, E3 +60629.323}
SPL {X  -160.000, Y  +518.188, Z    +0.000, E1   -14.845, E3 +60649.952}
SPL {X  -160.000, Y  +520.790, Z    +0.000, E1   -14.839, E3 +60670.781}
SPL {X  -160.000, Y  +523.469, Z    +0.000, E1   -14.855, E3 +60692.229}
SPL {X  -160.000, Y  +526.403, Z    +0.000, E1   -14.858, E3 +60715.766}
SPL {X  -160.000, Y  +529.266, Z    +0.000, E1   -14.848, E3 +60738.773}
SPL {X  -160.000, Y  +531.688, Z    +0.000, E1   -14.826, E3 +60758.323}
SPL {X  -160.000, Y  +534.214, Z    +0.000, E1   -14.841, E3 +60778.586}
SPL {X  -160.000, Y  +537.002, Z    +0.000, E1   -14.839, E3 +60801.004}
SPL {X  -160.000, Y  +539.729, Z    +0.000, E1   -14.840, E3 +60822.815}
SPL {X  -160.000, Y  +542.408, Z    +0.000, E1   -14.839, E3 +60844.368}
SPL {X  -160.000, Y  +545.014, Z    +0.000, E1   -14.831, E3 +60865.314}
SPL {X  -160.000, Y  +547.659, Z    +0.000, E1   -14.839, E3 +60886.528}
SPL {X  -160.000, Y  +550.215, Z    +0.000, E1   -14.827, E3 +60907.093}
SPL {X  -160.000, Y  +552.762, Z    +0.000, E1   -14.836, E3 +60927.511}
SPL {X  -160.000, Y  +555.331, Z    +0.000, E1   -14.837, E3 +60948.052}
SPL {X  -160.000, Y  +558.235, Z    +0.000, E1   -14.869, E3 +60971.216}
SPL {X  -160.000, Y  +561.088, Z    +0.000, E1   -14.848, E3 +60994.135}
SPL {X  -160.000, Y  +563.693, Z    +0.000, E1   -14.852, E3 +61014.995}
SPL {X  -160.000, Y  +566.560, Z    +0.000, E1   -14.865, E3 +61037.973}
SPL {X  -160.000, Y  +569.305, Z    +0.000, E1   -14.848, E3 +61060.001}
SPL {X  -160.000, Y  +571.769, Z    +0.000, E1   -14.852, E3 +61079.747}
SPL {X  -160.000, Y  +574.366, Z    +0.000, E1   -14.855, E3 +61100.534}
SPL {X  -160.000, Y  +577.037, Z    +0.000, E1   -14.859, E3 +61121.933}
SPL {X  -160.000, Y  +579.855, Z    +0.000, E1   -14.869, E3 +61144.461}
SPL {X  -160.000, Y  +582.456, Z    +0.000, E1   -14.854, E3 +61165.321}
SPL {X  -160.000, Y  +585.083, Z    +0.000, E1   -14.866, E3 +61186.370}
SPL {X  -160.000, Y  +587.675, Z    +0.000, E1   -14.853, E3 +61207.161}
SPL {X  -160.000, Y  +590.216, Z    +0.000, E1   -14.864, E3 +61227.480}
SPL {X  -160.000, Y  +592.848, Z    +0.000, E1   -14.865, E3 +61248.532}
SPL {X  -160.000, Y  +595.342, Z    +0.000, E1   -14.848, E3 +61268.709}
SPL {X  -160.000, Y  +597.995, Z    +0.000, E1   -14.848, E3 +61290.049}
SPL {X  -160.000, Y  +600.731, Z    +0.000, E1   -14.846, E3 +61312.001}
SPL {X  -160.000, Y  +603.404, Z    +0.000, E1   -14.846, E3 +61333.436}
SPL {X  -160.000, Y  +605.923, Z    +0.000, E1   -14.838, E3 +61353.677}
SPL {X  -160.000, Y  +608.492, Z    +0.000, E1   -14.846, E3 +61374.281}
SPL {X  -160.000, Y  +611.345, Z    +0.000, E1   -14.856, E3 +61397.139}
SPL {X  -160.000, Y  +614.087, Z    +0.000, E1   -14.839, E3 +61419.198}
SPL {X  -160.000, Y  +616.566, Z    +0.000, E1   -14.839, E3 +61439.092}
SPL {X  -160.000, Y  +619.350, Z    +0.000, E1   -14.855, E3 +61461.380}
SPL {X  -160.000, Y  +622.198, Z    +0.000, E1   -14.846, E3 +61484.265}
SPL {X  -160.000, Y  +624.642, Z    +0.000, E1   -14.829, E3 +61503.937}
SPL {X  -160.000, Y  +627.119, Z    +0.000, E1   -14.843, E3 +61523.777}
SPL {X  -160.000, Y  +629.682, Z    +0.000, E1   -14.838, E3 +61544.346}
SPL {X  -160.000, Y  +632.223, Z    +0.000, E1   -14.841, E3 +61564.737}
SPL {X  -160.000, Y  +634.941, Z    +0.000, E1   -14.846, E3 +61586.535}
SPL {X  -160.000, Y  +637.723, Z    +0.000, E1   -14.844, E3 +61608.879}
SPL {X  -160.000, Y  +640.315, Z    +0.000, E1   -14.836, E3 +61629.677}
SPL {X  -160.000, Y  +643.085, Z    +0.000, E1   -14.865, E3 +61651.728}
SPL {X  -160.000, Y  +645.845, Z    +0.000, E1   -14.848, E3 +61673.916}
SPL {X  -160.000, Y  +648.229, Z    +0.000, E1   -14.834, E3 +61693.126}
SPL {X  -160.000, Y  +650.656, Z    +0.000, E1   -14.835, E3 +61712.683}
SPL {X  -160.000, Y  +653.134, Z    +0.000, E1   -14.827, E3 +61732.610}
SPL {X  -160.000, Y  +655.670, Z    +0.000, E1   -14.841, E3 +61752.904}
SPL {X  -160.000, Y  +658.349, Z    +0.000, E1   -14.842, E3 +61774.379}
SPL {X  -160.000, Y  +660.936, Z    +0.000, E1   -14.838, E3 +61795.131}
SPL {X  -160.000, Y  +663.567, Z    +0.000, E1   -14.845, E3 +61816.262}
SPL {X  -160.000, Y  +666.216, Z    +0.000, E1   -14.832, E3 +61837.578}
SPL {X  -159.997, Y  +668.731, Z    +0.000, E1   -14.834, E3 +61857.770}
SPL {X  -159.962, Y  +671.176, Z    +0.000, E1   -14.822, E3 +61877.481}
SPL {X  -159.895, Y  +673.507, Z    +0.000, E1   -14.821, E3 +61896.213}
SPL {X  -159.785, Y  +675.985, Z    +0.000, E1   -14.818, E3 +61916.214}
SPL {X  -159.627, Y  +678.622, Z    +0.000, E1   -14.804, E3 +61937.567}
SPL {X  -159.438, Y  +681.094, Z    +0.000, E1   -14.770, E3 +61957.738}
SPL {X  -159.262, Y  +683.054, Z    +0.000, E1   -14.719, E3 +61973.967}
ENDSPLINE

SPLINE
SPL {X  -159.661, Y  +678.114, Z    +0.000, E1    -9.575, E3 +62003.559}
SPL {X  -159.942, Y  +672.020, Z    +0.000, E1    -4.692, E3 +62022.185}
SPL {X  -160.000, Y  +664.971, Z    +0.000, E1    +0.516, E3 +62041.736}
SPL {X  -160.000, Y  +660.032, Z    +0.000, E1    +3.995, E3 +62053.679}
SPL {X  -160.000, Y  +652.280, Z    +0.000, E1    +8.913, E3 +62072.194}
SPL {X  -160.000, Y  +644.147, Z    +0.000, E1   +13.158, E3 +62095.744}
SPL {X  -160.000, Y  +641.594, Z    +0.000, E1   +13.488, E3 +62114.185}
SPL {X  -160.000, Y  +639.799, Z    +0.000, E1   +13.486, E3 +62130.095}
SPL {X  -160.000, Y  +637.896, Z    +0.000, E1   +13.493, E3 +62146.910}
SPL {X  -160.000, Y  +635.832, Z    +0.000, E1   +13.499, E3 +62165.169}
SPL {X  -160.000, Y  +633.839, Z    +0.000, E1   +13.489, E3 +62182.858}
SPL {X  -160.000, Y  +631.625, Z    +0.000, E1   +13.508, E3 +62202.398}
SPL {X  -160.000, Y  +629.417, Z    +0.000, E1   +13.491, E3 +62222.010}
SPL {X  -160.000, Y  +627.180, Z    +0.000, E1   +13.508, E3 +62241.764}
SPL {X  -160.000, Y  +624.970, Z    +0.000, E1   +13.490, E3 +62261.414}
SPL {X  -160.000, Y  +623.020, Z    +0.000, E1   +13.491, E3 +62278.644}
SPL {X  -160.000, Y  +620.888, Z    +0.000, E1   +13.501, E3 +62297.506}
SPL {X  -160.000, Y  +618.790, Z    +0.000, E1   +13.488, E3 +62316.129}
SPL {X  -160.000, Y  +616.631, Z    +0.000, E1   +13.504, E3 +62335.182}
SPL {X  -160.000, Y  +614.230, Z    +0.000, E1   +13.510, E3 +62356.378}
SPL {X  -160.000, Y  +612.132, Z    +0.000, E1   +13.485, E3 +62375.094}
SPL {X  -160.000, Y  +610.405, Z    +0.000, E1   +13.477, E3 +62390.468}
SPL {X  -160.000, Y  +608.437, Z    +0.000, E1   +13.502, E3 +62407.723}
SPL {X  -160.000, Y  +606.281, Z    +0.000, E1   +13.502, E3 +62426.741}
SPL {X  -160.000, Y  +604.124, Z    +0.000, E1   +13.513, E3 +62445.796}
SPL {X  -160.000, Y  +601.878, Z    +0.000, E1   +13.505, E3 +62465.693}
SPL {X  -160.000, Y  +599.648, Z    +0.000, E1   +13.506, E3 +62485.470}
SPL {X  -160.000, Y  +597.673, Z    +0.000, E1   +13.479, E3 +62503.143}
SPL {X  -160.000, Y  +595.601, Z    +0.000, E1   +13.499, E3 +62521.427}
SPL {X  -160.000, Y  +593.187, Z    +0.000, E1   +13.500, E3 +62542.807}
SPL {X  -160.000, Y  +591.079, Z    +0.000, E1   +13.483, E3 +62561.533}
SPL {X  -160.000, Y  +589.151, Z    +0.000, E1   +13.489, E3 +62578.584}
SPL {X  -160.000, Y  +586.908, Z    +0.000, E1   +13.501, E3 +62598.429}
SPL {X  -160.000, Y  +584.660, Z    +0.000, E1   +13.490, E3 +62618.371}
SPL {X  -160.000, Y  +582.409, Z    +0.000, E1   +13.499, E3 +62638.289}
SPL {X  -160.000, Y  +580.150, Z    +0.000, E1   +13.490, E3 +62658.336}
SPL {X  -160.000, Y  +577.953, Z    +0.000, E1   +13.493, E3 +62677.794}
SPL {X  -160.000, Y  +575.630, Z    +0.000, E1   +13.502, E3 +62698.278}
SPL {X  -160.000, Y  +573.418, Z    +0.000, E1   +13.502, E3 +62717.786}
SPL {X  -160.000, Y  +571.226, Z    +0.000, E1   +13.520, E3 +62736.995}
SPL {X  -160.000, Y  +569.166, Z    +0.000, E1   +13.512, E3 +62755.185}
SPL {X  -160.000, Y  +567.275, Z    +0.000, E1   +13.517, E3 +62771.852}
SPL {X  -160.000, Y  +565.259, Z    +0.000, E1   +13.523, E3 +62789.641}
SPL {X  -160.000, Y  +563.305, Z    +0.000, E1   +13.512, E3 +62806.980}
SPL {X  -160.000, Y  +561.240, Z    +0.000, E1   +13.521, E3 +62825.241}
SPL {X  -160.000, Y  +558.881, Z    +0.000, E1   +13.524, E3 +62846.084}
SPL {X  -160.000, Y  +556.697, Z    +0.000, E1   +13.510, E3 +62865.470}
SPL {X  -160.000, Y  +554.624, Z    +0.000, E1   +13.512, E3 +62883.801}
SPL {X  -160.000, Y  +552.465, Z    +0.000, E1   +13.514, E3 +62902.885}
SPL {X  -160.000, Y  +550.315, Z    +0.000, E1   +13.514, E3 +62921.879}
SPL {X  -160.000, Y  +548.056, Z    +0.000, E1   +13.519, E3 +62941.880}
SPL {X  -160.000, Y  +545.826, Z    +0.000, E1   +13.501, E3 +62961.757}
SPL {X  -160.000, Y  +543.677, Z    +0.000, E1   +13.502, E3 +62980.815}
SPL {X  -160.000, Y  +541.664, Z    +0.000, E1   +13.489, E3 +62998.700}
SPL {X  -160.000, Y  +539.659, Z    +0.000, E1   +13.494, E3 +63016.461}
SPL {X  -160.000, Y  +537.370, Z    +0.000, E1   +13.501, E3 +63036.700}
SPL {X  -160.000, Y  +535.056, Z    +0.000, E1   +13.506, E3 +63057.095}
SPL {X  -160.000, Y  +532.975, Z    +0.000, E1   +13.494, E3 +63075.582}
SPL {X  -160.000, Y  +530.925, Z    +0.000, E1   +13.499, E3 +63093.744}
SPL {X  -160.000, Y  +528.768, Z    +0.000, E1   +13.498, E3 +63112.845}
SPL {X  -160.000, Y  +526.547, Z    +0.000, E1   +13.499, E3 +63132.514}
SPL {X  -160.000, Y  +523.964, Z    +0.000, E1   +13.742, E3 +63152.018}
SPL {X  -160.000, Y  +513.971, Z    +0.000, E1   +18.644, E3 +63170.930}
SPL {X  -160.000, Y  +513.562, Z    +0.000, E1   +16.972, E3 +63190.807}
SPL {X  -160.000, Y  +513.358, Z    +0.000, E1   +15.267, E3 +63211.079}
SPL {X  -160.000, Y  +512.244, Z    +0.000, E1   +14.473, E3 +63229.535}
SPL {X  -160.000, Y  +509.675, Z    +0.000, E1   +14.481, E3 +63250.679}
SPL {X  -160.000, Y  +507.162, Z    +0.000, E1   +14.470, E3 +63271.419}
SPL {X  -160.000, Y  +504.735, Z    +0.000, E1   +14.473, E3 +63291.390}
SPL {X  -160.000, Y  +502.261, Z    +0.000, E1   +14.476, E3 +63311.726}
SPL {X  -160.000, Y  +499.798, Z    +0.000, E1   +14.482, E3 +63331.928}
SPL {X  -160.000, Y  +497.435, Z    +0.000, E1   +14.476, E3 +63351.405}
SPL {X  -160.000, Y  +495.089, Z    +0.000, E1   +14.475, E3 +63370.772}
SPL {X  -160.000, Y  +492.764, Z    +0.000, E1   +14.469, E3 +63389.943}
SPL {X  -160.000, Y  +490.292, Z    +0.000, E1   +14.476, E3 +63410.344}
SPL {X  -160.000, Y  +487.641, Z    +0.000, E1   +14.470, E3 +63432.240}
SPL {X  -160.000, Y  +485.054, Z    +0.000, E1   +14.460, E3 +63453.683}
SPL {X  -160.000, Y  +482.421, Z    +0.000, E1   +14.461, E3 +63475.401}
SPL {X  -160.000, Y  +480.000, Z    +0.000, E1   +14.451, E3 +63495.366}
SPL {X  -160.000, Y  +477.551, Z    +0.000, E1   +14.466, E3 +63515.494}
SPL {X  -160.000, Y  +475.253, Z    +0.000, E1   +14.450, E3 +63534.468}
SPL {X  -160.000, Y  +473.070, Z    +0.000, E1   +14.454, E3 +63552.489}
SPL {X  -160.000, Y  +470.603, Z    +0.000, E1   +14.464, E3 +63572.789}
SPL {X  -160.000, Y  +468.243, Z    +0.000, E1   +14.458, E3 +63592.189}
SPL {X  -160.000, Y  +465.791, Z    +0.000, E1   +14.475, E3 +63612.333}
SPL {X  -160.000, Y  +463.103, Z    +0.000, E1   +14.474, E3 +63634.481}
SPL {X  -160.000, Y  +460.743, Z    +0.000, E1   +14.465, E3 +63653.890}
SPL {X  -160.000, Y  +458.292, Z    +0.000, E1   +14.492, E3 +63673.889}
SPL {X  -160.000, Y  +455.874, Z    +0.000, E1   +14.484, E3 +63693.747}
SPL {X  -160.000, Y  +453.555, Z    +0.000, E1   +14.488, E3 +63712.826}
SPL {X  -160.000, Y  +451.093, Z    +0.000, E1   +14.485, E3 +63733.138}
SPL {X  -160.000, Y  +448.700, Z    +0.000, E1   +14.483, E3 +63752.827}
SPL {X  -160.000, Y  +446.277, Z    +0.000, E1   +14.485, E3 +63772.751}
SPL {X  -160.000, Y  +443.879, Z    +0.000, E1   +14.485, E3 +63792.489}
SPL {X  -160.000, Y  +441.447, Z    +0.000, E1   +14.485, E3 +63812.496}
SPL {X  -160.000, Y  +439.006, Z    +0.000, E1   +14.488, E3 +63832.579}
SPL {X  -160.000, Y  +436.311, Z    +0.000, E1   +14.498, E3 +63854.738}
SPL {X  -160.000, Y  +433.559, Z    +0.000, E1   +14.491, E3 +63877.408}
SPL {X  -160.000, Y  +431.162, Z    +0.000, E1   +14.479, E3 +63897.159}
SPL {X  -160.000, Y  +429.152, Z    +0.000, E1   +14.469, E3 +63913.740}
SPL {X  -160.000, Y  +426.863, Z    +0.000, E1   +14.490, E3 +63932.519}
SPL {X  -160.000, Y  +424.653, Z    +0.000, E1   +14.467, E3 +63950.779}
SPL {X  -160.000, Y  +422.337, Z    +0.000, E1   +14.492, E3 +63969.763}
SPL {X  -160.000, Y  +419.639, Z    +0.000, E1   +14.504, E3 +63991.803}
SPL {X  -160.000, Y  +417.127, Z    +0.000, E1   +14.501, E3 +64012.394}
SPL {X  -160.000, Y  +414.849, Z    +0.000, E1   +14.496, E3 +64031.128}
SPL {X  -160.000, Y  +412.396, Z    +0.000, E1   +14.505, E3 +64051.317}
SPL {X  -160.000, Y  +409.815, Z    +0.000, E1   +14.498, E3 +64072.571}
SPL {X  -160.000, Y  +407.614, Z    +0.000, E1   +14.484, E3 +64090.697}
SPL {X  -160.000, Y  +405.406, Z    +0.000, E1   +14.501, E3 +64108.760}
SPL {X  -160.000, Y  +402.958, Z    +0.000, E1   +14.500, E3 +64128.930}
SPL {X  -160.000, Y  +400.690, Z    +0.000, E1   +14.484, E3 +64147.641}
SPL {X  -160.000, Y  +398.391, Z    +0.000, E1   +14.502, E3 +64166.467}
SPL {X  -160.000, Y  +395.999, Z    +0.000, E1   +14.484, E3 +64186.257}
SPL {X  -160.000, Y  +393.685, Z    +0.000, E1   +14.486, E3 +64205.330}
SPL {X  -159.999, Y  +391.313, Z    +0.000, E1   +14.479, E3 +64224.912}
SPL {X  -159.970, Y  +388.900, Z    +0.000, E1   +14.480, E3 +64244.796}
SPL {X  -159.903, Y  +386.417, Z    +0.000, E1   +14.475, E3 +64265.301}
SPL {X  -159.796, Y  +383.921, Z    +0.000, E1   +14.466, E3 +64285.957}
SPL {X  -159.651, Y  +381.443, Z    +0.000, E1   +14.453, E3 +64306.504}
SPL {X  -159.474, Y  +379.042, Z    +0.000, E1   +14.434, E3 +64326.468}
SPL {X  -159.316, Y  +377.219, Z    +0.000, E1   +14.400, E3 +64341.697}
ENDSPLINE

SPLINE
SPL {X  -159.452, Y  +378.767, Z    +0.000, E1   +11.887, E3 +64362.686}
SPL {X  -159.840, Y  +384.856, Z    +0.000, E1    +7.126, E3 +64381.657}
SPL {X  -159.991, Y  +390.336, Z    +0.000, E1    +2.803, E3 +64395.480}
SPL {X  -160.000, Y  +403.532, Z    +0.000, E1    -6.523, E3 +64413.201}
SPL {X  -160.000, Y  +409.023, Z    +0.000, E1   -10.003, E3 +64423.975}
SPL {X  -160.000, Y  +418.032, Z    +0.000, E1   -14.569, E3 +64448.834}
SPL {X  -160.000, Y  +420.561, Z    +0.000, E1   -14.816, E3 +64466.314}
SPL {X  -160.000, Y  +422.801, Z    +0.000, E1   -14.823, E3 +64484.262}
SPL {X  -160.000, Y  +425.518, Z    +0.000, E1   -14.845, E3 +64506.037}
SPL {X  -160.000, Y  +428.688, Z    +0.000, E1   -14.854, E3 +64531.445}
SPL {X  -160.000, Y  +431.971, Z    +0.000, E1   -14.849, E3 +64557.914}
SPL {X  -160.000, Y  +435.345, Z    +0.000, E1   -14.857, E3 +64584.964}
SPL {X  -160.000, Y  +438.732, Z    +0.000, E1   -14.858, E3 +64612.112}
SPL {X  -160.000, Y  +441.925, Z    +0.000, E1   -14.848, E3 +64637.783}
SPL {X  -160.000, Y  +444.299, Z    +0.000, E1   -14.809, E3 +64656.967}
SPL {X  -160.000, Y  +446.229, Z    +0.000, E1   -14.820, E3 +64672.386}
SPL {X  -160.000, Y  +448.987, Z    +0.000, E1   -14.868, E3 +64694.323}
SPL {X  -160.000, Y  +452.351, Z    +0.000, E1   -14.871, E3 +64721.299}
SPL {X  -160.000, Y  +455.709, Z    +0.000, E1   -14.880, E3 +64748.113}
SPL {X  -160.000, Y  +458.189, Z    +0.000, E1   -14.832, E3 +64768.115}
SPL {X  -160.000, Y  +459.885, Z    +0.000, E1   -14.825, E3 +64781.785}
SPL {X  -160.000, Y  +462.438, Z    +0.000, E1   -14.868, E3 +64802.195}
SPL {X  -160.000, Y  +465.575, Z    +0.000, E1   -14.849, E3 +64827.504}
SPL {X  -160.000, Y  +468.581, Z    +0.000, E1   -14.841, E3 +64851.736}
SPL {X  -160.000, Y  +471.795, Z    +0.000, E1   -14.854, E3 +64877.523}
SPL {X  -160.000, Y  +475.138, Z    +0.000, E1   -14.853, E3 +64904.374}
SPL {X  -160.000, Y  +477.981, Z    +0.000, E1   -14.823, E3 +64927.294}
SPL {X  -160.000, Y  +480.658, Z    +0.000, E1   -14.835, E3 +64948.770}
SPL {X  -160.000, Y  +483.534, Z    +0.000, E1   -14.838, E3 +64971.865}
SPL {X  -160.000, Y  +486.226, Z    +0.000, E1   -14.823, E3 +64993.530}
SPL {X  -160.000, Y  +488.751, Z    +0.000, E1   -14.827, E3 +65013.802}
SPL {X  -160.000, Y  +491.612, Z    +0.000, E1   -14.844, E3 +65036.725}
SPL {X  -160.000, Y  +494.417, Z    +0.000, E1   -14.827, E3 +65059.316}
SPL {X  -160.000, Y  +496.961, Z    +0.000, E1   -14.824, E3 +65079.760}
SPL {X  -160.000, Y  +499.610, Z    +0.000, E1   -14.830, E3 +65101.032}
SPL {X  -160.000, Y  +502.268, Z    +0.000, E1   -14.832, E3 +65122.302}
SPL {X  -160.000, Y  +505.041, Z    +0.000, E1   -14.849, E3 +65144.464}
SPL {X  -160.000, Y  +507.743, Z    +0.000, E1   -14.842, E3 +65166.088}
SPL {X  -160.000, Y  +510.437, Z    +0.000, E1   -14.860, E3 +65187.602}
SPL {X  -160.000, Y  +513.179, Z    +0.000, E1   -14.849, E3 +65209.649}
SPL {X  -160.000, Y  +515.613, Z    +0.000, E1   -14.829, E3 +65229.320}
SPL {X  -160.000, Y  +518.188, Z    +0.000, E1   -14.845, E3 +65249.949}
SPL {X  -160.000, Y  +520.790, Z    +0.000, E1   -14.839, E3 +65270.778}
SPL {X  -160.000, Y  +523.469, Z    +0.000, E1   -14.855, E3 +65292.226}
SPL {X  -160.000, Y  +526.403, Z    +0.000, E1   -14.858, E3 +65315.762}
SPL {X  -160.000, Y  +529.266, Z    +0.000, E1   -14.848, E3 +65338.770}
SPL {X  -160.000, Y  +531.688, Z    +0.000, E1   -14.826, E3 +65358.319}
SPL {X  -160.000, Y  +534.214, Z    +0.000, E1   -14.841, E3 +65378.582}
SPL {X  -160.000, Y  +537.002, Z    +0.000, E1   -14.839, E3 +65401.001}
SPL {X  -160.000, Y  +539.729, Z    +0.000, E1   -14.840, E3 +65422.812}
SPL {X  -160.000, Y  +542.408, Z    +0.000, E1   -14.839, E3 +65444.365}
SPL {X  -160.000, Y  +545.014, Z    +0.000, E1   -14.831, E3 +65465.310}
SPL {X  -160.000, Y  +547.659, Z    +0.000, E1   -14.839, E3 +65486.525}
SPL {X  -160.000, Y  +550.215, Z    +0.000, E1   -14.827, E3 +65507.090}
SPL {X  -160.000, Y  +552.762, Z    +0.000, E1   -14.836, E3 +65527.508}
SPL {X  -160.000, Y  +555.331, Z    +0.000, E1   -14.837, E3 +65548.049}
SPL {X  -160.000, Y  +558.235, Z    +0.000, E1   -14.869, E3 +65571.213}
SPL {X  -160.000, Y  +561.088, Z    +0.000, E1   -14.848, E3 +65594.131}
SPL {X  -160.000, Y  +563.693, Z    +0.000, E1   -14.852, E3 +65614.992}
SPL {X  -160.000, Y  +566.560, Z    +0.000, E1   -14.865, E3 +65637.969}
SPL {X  -160.000, Y  +569.305, Z    +0.000, E1   -14.848, E3 +65659.998}
SPL {X  -160.000, Y  +571.769, Z    +0.000, E1   -14.852, E3 +65679.744}
SPL {X  -160.000, Y  +574.366, Z    +0.000, E1   -14.855, E3 +65700.531}
SPL {X  -160.000, Y  +577.037, Z    +0.000, E1   -14.859, E3 +65721.930}
SPL {X  -160.000, Y  +579.855, Z    +0.000, E1   -14.869, E3 +65744.457}
SPL {X  -160.000, Y  +582.456, Z    +0.000, E1   -14.854, E3 +65765.317}
SPL {X  -160.000, Y  +585.083, Z    +0.000, E1   -14.866, E3 +65786.367}
SPL {X  -160.000, Y  +587.675, Z    +0.000, E1   -14.853, E3 +65807.158}
SPL {X  -160.000, Y  +590.216, Z    +0.000, E1   -14.864, E3 +65827.477}
SPL {X  -160.000, Y  +592.848, Z    +0.000, E1   -14.865, E3 +65848.528}
SPL {X  -160.000, Y  +595.342, Z    +0.000, E1   -14.848, E3 +65868.706}
SPL {X  -160.000, Y  +597.995, Z    +0.000, E1   -14.848, E3 +65890.046}
SPL {X  -160.000, Y  +600.731, Z    +0.000, E1   -14.846, E3 +65911.997}
SPL {X  -160.000, Y  +603.404, Z    +0.000, E1   -14.846, E3 +65933.433}
SPL {X  -160.000, Y  +605.923, Z    +0.000, E1   -14.838, E3 +65953.674}
SPL {X  -160.000, Y  +608.492, Z    +0.000, E1   -14.846, E3 +65974.278}
SPL {X  -160.000, Y  +611.345, Z    +0.000, E1   -14.856, E3 +65997.136}
SPL {X  -160.000, Y  +614.087, Z    +0.000, E1   -14.839, E3 +66019.195}
SPL {X  -160.000, Y  +616.566, Z    +0.000, E1   -14.839, E3 +66039.089}
SPL {X  -160.000, Y  +619.350, Z    +0.000, E1   -14.855, E3 +66061.377}
SPL {X  -160.000, Y  +622.198, Z    +0.000, E1   -14.846, E3 +66084.262}
SPL {X  -160.000, Y  +624.642, Z    +0.000, E1   -14.829, E3 +66103.934}
SPL {X  -160.000, Y  +627.119, Z    +0.000, E1   -14.843, E3 +66123.774}
SPL {X  -160.000, Y  +629.682, Z    +0.000, E1   -14.838, E3 +66144.343}
SPL {X  -160.000, Y  +632.223, Z    +0.000, E1   -14.841, E3 +66164.734}
SPL {X  -160.000, Y  +634.941, Z    +0.000, E1   -14.846, E3 +66186.532}
SPL {X  -160.000, Y  +637.723, Z    +0.000, E1   -14.844, E3 +66208.876}
SPL {X  -160.000, Y  +640.315, Z    +0.000, E1   -14.836, E3 +66229.674}
SPL {X  -160.000, Y  +643.085, Z    +0.000, E1   -14.865, E3 +66251.725}
SPL {X  -160.000, Y  +645.845, Z    +0.000, E1   -14.848, E3 +66273.913}
SPL {X  -160.000, Y  +648.229, Z    +0.000, E1   -14.834, E3 +66293.123}
SPL {X  -160.000, Y  +650.656, Z    +0.000, E1   -14.835, E3 +66312.679}
SPL {X  -160.000, Y  +653.134, Z    +0.000, E1   -14.827, E3 +66332.606}
SPL {X  -160.000, Y  +655.670, Z    +0.000, E1   -14.841, E3 +66352.901}
SPL {X  -160.000, Y  +658.349, Z    +0.000, E1   -14.842, E3 +66374.376}
SPL {X  -160.000, Y  +660.936, Z    +0.000, E1   -14.838, E3 +66395.128}
SPL {X  -160.000, Y  +663.567, Z    +0.000, E1   -14.845, E3 +66416.258}
SPL {X  -160.000, Y  +666.216, Z    +0.000, E1   -14.832, E3 +66437.575}
SPL {X  -159.997, Y  +668.731, Z    +0.000, E1   -14.834, E3 +66457.767}
SPL {X  -159.962, Y  +671.176, Z    +0.000, E1   -14.822, E3 +66477.478}
SPL {X  -159.895, Y  +673.507, Z    +0.000, E1   -14.821, E3 +66496.209}
SPL {X  -159.785, Y  +675.985, Z    +0.000, E1   -14.818, E3 +66516.211}
SPL {X  -159.627, Y  +678.622, Z    +0.000, E1   -14.804, E3 +66537.564}
SPL {X  -159.438, Y  +681.094, Z    +0.000, E1   -14.770, E3 +66557.735}
SPL {X  -159.262, Y  +683.054, Z    +0.000, E1   -14.719, E3 +66573.964}
ENDSPLINE

SPLINE
SPL {X  -159.661, Y  +678.114, Z    +0.000, E1    -9.575, E3 +66603.555}
SPL {X  -159.942, Y  +672.020, Z    +0.000, E1    -4.692, E3 +66622.182}
SPL {X  -160.000, Y  +664.971, Z    +0.000, E1    +0.516, E3 +66641.733}
SPL {X  -160.000, Y  +660.032, Z    +0.000, E1    +3.995, E3 +66653.675}
SPL {X  -160.000, Y  +652.280, Z    +0.000, E1    +8.913, E3 +66672.190}
SPL {X  -160.000, Y  +644.147, Z    +0.000, E1   +13.158, E3 +66695.741}
SPL {X  -160.000, Y  +641.594, Z    +0.000, E1   +13.488, E3 +66714.182}
SPL {X  -160.000, Y  +639.799, Z    +0.000, E1   +13.486, E3 +66730.092}
SPL {X  -160.000, Y  +637.896, Z    +0.000, E1   +13.493, E3 +66746.907}
SPL {X  -160.000, Y  +635.832, Z    +0.000, E1   +13.499, E3 +66765.166}
SPL {X  -160.000, Y  +633.839, Z    +0.000, E1   +13.489, E3 +66782.854}
SPL {X  -160.000, Y  +631.625, Z    +0.000, E1   +13.508, E3 +66802.395}
SPL {X  -160.000, Y  +629.417, Z    +0.000, E1   +13.491, E3 +66822.007}
SPL {X  -160.000, Y  +627.180, Z    +0.000, E1   +13.508, E3 +66841.761}
SPL {X  -160.000, Y  +624.970, Z    +0.000, E1   +13.490, E3 +66861.411}
SPL {X  -160.000, Y  +623.020, Z    +0.000, E1   +13.491, E3 +66878.640}
SPL {X  -160.000, Y  +620.888, Z    +0.000, E1   +13.501, E3 +66897.503}
SPL {X  -160.000, Y  +618.790, Z    +0.000, E1   +13.488, E3 +66916.125}
SPL {X  -160.000, Y  +616.631, Z    +0.000, E1   +13.504, E3 +66935.179}
SPL {X  -160.000, Y  +614.230, Z    +0.000, E1   +13.510, E3 +66956.375}
SPL {X  -160.000, Y  +612.132, Z    +0.000, E1   +13.485, E3 +66975.091}
SPL {X  -160.000, Y  +610.405, Z    +0.000, E1   +13.477, E3 +66990.464}
SPL {X  -160.000, Y  +608.437, Z    +0.000, E1   +13.502, E3 +67007.720}
SPL {X  -160.000, Y  +606.281, Z    +0.000, E1   +13.502, E3 +67026.737}
SPL {X  -160.000, Y  +604.124, Z    +0.000, E1   +13.513, E3 +67045.793}
SPL {X  -160.000, Y  +601.878, Z    +0.000, E1   +13.505, E3 +67065.690}
SPL {X  -160.000, Y  +599.648, Z    +0.000, E1   +13.506, E3 +67085.467}
SPL {X  -160.000, Y  +597.673, Z    +0.000, E1   +13.479, E3 +67103.140}
SPL {X  -160.000, Y  +595.601, Z    +0.000, E1   +13.499, E3 +67121.423}
SPL {X  -160.000, Y  +593.187, Z    +0.000, E1   +13.500, E3 +67142.803}
SPL {X  -160.000, Y  +591.079, Z    +0.000, E1   +13.483, E3 +67161.530}
SPL {X  -160.000, Y  +589.151, Z    +0.000, E1   +13.489, E3 +67178.581}
SPL {X  -160.000, Y  +586.908, Z    +0.000, E1   +13.501, E3 +67198.426}
SPL {X  -160.000, Y  +584.660, Z    +0.000, E1   +13.490, E3 +67218.368}
SPL {X  -160.000, Y  +582.409, Z    +0.000, E1   +13.499, E3 +67238.286}
SPL {X  -160.000, Y  +580.150, Z    +0.000, E1   +13.490, E3 +67258.332}
SPL {X  -160.000, Y  +577.953, Z    +0.000, E1   +13.493, E3 +67277.791}
SPL {X  -160.000, Y  +575.630, Z    +0.000, E1   +13.502, E3 +67298.275}
SPL {X  -160.000, Y  +573.418, Z    +0.000, E1   +13.502, E3 +67317.783}
SPL {X  -160.000, Y  +571.226, Z    +0.000, E1   +13.520, E3 +67336.991}
SPL {X  -160.000, Y  +569.166, Z    +0.000, E1   +13.512, E3 +67355.182}
SPL {X  -160.000, Y  +567.275, Z    +0.000, E1   +13.517, E3 +67371.849}
SPL {X  -160.000, Y  +565.259, Z    +0.000, E1   +13.523, E3 +67389.638}
SPL {X  -160.000, Y  +563.305, Z    +0.000, E1   +13.512, E3 +67406.977}
SPL {X  -160.000, Y  +561.240, Z    +0.000, E1   +13.521, E3 +67425.238}
SPL {X  -160.000, Y  +558.881, Z    +0.000, E1   +13.524, E3 +67446.081}
SPL {X  -160.000, Y  +556.697, Z    +0.000, E1   +13.510, E3 +67465.467}
SPL {X  -160.000, Y  +554.624, Z    +0.000, E1   +13.512, E3 +67483.797}
SPL {X  -160.000, Y  +552.465, Z    +0.000, E1   +13.514, E3 +67502.882}
SPL {X  -160.000, Y  +550.315, Z    +0.000, E1   +13.514, E3 +67521.875}
SPL {X  -160.000, Y  +548.056, Z    +0.000, E1   +13.519, E3 +67541.876}
SPL {X  -160.000, Y  +545.826, Z    +0.000, E1   +13.501, E3 +67561.754}
SPL {X  -160.000, Y  +543.677, Z    +0.000, E1   +13.502, E3 +67580.812}
SPL {X  -160.000, Y  +541.664, Z    +0.000, E1   +13.489, E3 +67598.697}
SPL {X  -160.000, Y  +539.659, Z    +0.000, E1   +13.494, E3 +67616.457}
SPL {X  -160.000, Y  +537.370, Z    +0.000, E1   +13.501, E3 +67636.696}
SPL {X  -160.000, Y  +535.056, Z    +0.000, E1   +13.506, E3 +67657.092}
SPL {X  -160.000, Y  +532.975, Z    +0.000, E1   +13.494, E3 +67675.579}
SPL {X  -160.000, Y  +530.925, Z    +0.000, E1   +13.499, E3 +67693.740}
SPL {X  -160.000, Y  +528.768, Z    +0.000, E1   +13.498, E3 +67712.842}
SPL {X  -160.000, Y  +526.547, Z    +0.000, E1   +13.499, E3 +67732.510}
SPL {X  -160.000, Y  +523.964, Z    +0.000, E1   +13.742, E3 +67752.015}
SPL {X  -160.000, Y  +513.971, Z    +0.000, E1   +18.644, E3 +67770.927}
SPL {X  -160.000, Y  +513.562, Z    +0.000, E1   +16.972, E3 +67790.804}
SPL {X  -160.000, Y  +513.358, Z    +0.000, E1   +15.267, E3 +67811.076}
SPL {X  -160.000, Y  +512.244, Z    +0.000, E1   +14.473, E3 +67829.532}
SPL {X  -160.000, Y  +509.675, Z    +0.000, E1   +14.481, E3 +67850.675}
SPL {X  -160.000, Y  +507.162, Z    +0.000, E1   +14.470, E3 +67871.416}
SPL {X  -160.000, Y  +504.735, Z    +0.000, E1   +14.473, E3 +67891.387}
SPL {X  -160.000, Y  +502.261, Z    +0.000, E1   +14.476, E3 +67911.723}
SPL {X  -160.000, Y  +499.798, Z    +0.000, E1   +14.482, E3 +67931.925}
SPL {X  -160.000, Y  +497.435, Z    +0.000, E1   +14.476, E3 +67951.402}
SPL {X  -160.000, Y  +495.089, Z    +0.000, E1   +14.475, E3 +67970.769}
SPL {X  -160.000, Y  +492.764, Z    +0.000, E1   +14.469, E3 +67989.940}
SPL {X  -160.000, Y  +490.292, Z    +0.000, E1   +14.476, E3 +68010.341}
SPL {X  -160.000, Y  +487.641, Z    +0.000, E1   +14.470, E3 +68032.237}
SPL {X  -160.000, Y  +485.054, Z    +0.000, E1   +14.460, E3 +68053.680}
SPL {X  -160.000, Y  +482.421, Z    +0.000, E1   +14.461, E3 +68075.398}
SPL {X  -160.000, Y  +480.000, Z    +0.000, E1   +14.451, E3 +68095.362}
SPL {X  -160.000, Y  +477.551, Z    +0.000, E1   +14.466, E3 +68115.491}
SPL {X  -160.000, Y  +475.253, Z    +0.000, E1   +14.450, E3 +68134.465}
SPL {X  -160.000, Y  +473.070, Z    +0.000, E1   +14.454, E3 +68152.486}
SPL {X  -160.000, Y  +470.603, Z    +0.000, E1   +14.464, E3 +68172.786}
SPL {X  -160.000, Y  +468.243, Z    +0.000, E1   +14.458, E3 +68192.185}
SPL {X  -160.000, Y  +465.791, Z    +0.000, E1   +14.475, E3 +68212.330}
SPL {X  -160.000, Y  +463.103, Z    +0.000, E1   +14.474, E3 +68234.478}
SPL {X  -160.000, Y  +460.743, Z    +0.000, E1   +14.465, E3 +68253.887}
SPL {X  -160.000, Y  +458.292, Z    +0.000, E1   +14.492, E3 +68273.886}
SPL {X  -160.000, Y  +455.874, Z    +0.000, E1   +14.484, E3 +68293.743}
SPL {X  -160.000, Y  +453.555, Z    +0.000, E1   +14.488, E3 +68312.823}
SPL {X  -160.000, Y  +451.093, Z    +0.000, E1   +14.485, E3 +68333.135}
SPL {X  -160.000, Y  +448.700, Z    +0.000, E1   +14.483, E3 +68352.824}
SPL {X  -160.000, Y  +446.277, Z    +0.000, E1   +14.485, E3 +68372.748}
SPL {X  -160.000, Y  +443.879, Z    +0.000, E1   +14.485, E3 +68392.486}
SPL {X  -160.000, Y  +441.447, Z    +0.000, E1   +14.485, E3 +68412.493}
SPL {X  -160.000, Y  +439.006, Z    +0.000, E1   +14.488, E3 +68432.576}
SPL {X  -160.000, Y  +436.311, Z    +0.000, E1   +14.498, E3 +68454.735}
SPL {X  -160.000, Y  +433.559, Z    +0.000, E1   +14.491, E3 +68477.405}
SPL {X  -160.000, Y  +431.162, Z    +0.000, E1   +14.479, E3 +68497.156}
SPL {X  -160.000, Y  +429.152, Z    +0.000, E1   +14.469, E3 +68513.737}
SPL {X  -160.000, Y  +426.863, Z    +0.000, E1   +14.490, E3 +68532.516}
SPL {X  -160.000, Y  +424.653, Z    +0.000, E1   +14.467, E3 +68550.776}
SPL {X  -160.000, Y  +422.337, Z    +0.000, E1   +14.492, E3 +68569.760}
SPL {X  -160.000, Y  +419.639, Z    +0.000, E1   +14.504, E3 +68591.800}
SPL {X  -160.000, Y  +417.127, Z    +0.000, E1   +14.501, E3 +68612.391}
SPL {X  -160.000, Y  +414.849, Z    +0.000, E1   +14.496, E3 +68631.125}
SPL {X  -160.000, Y  +412.396, Z    +0.000, E1   +14.505, E3 +68651.314}
SPL {X  -160.000, Y  +409.815, Z    +0.000, E1   +14.498, E3 +68672.568}
SPL {X  -160.000, Y  +407.614, Z    +0.000, E1   +14.484, E3 +68690.693}
SPL {X  -160.000, Y  +405.406, Z    +0.000, E1   +14.501, E3 +68708.756}
SPL {X  -160.000, Y  +402.958, Z    +0.000, E1   +14.500, E3 +68728.927}
SPL {X  -160.000, Y  +400.690, Z    +0.000, E1   +14.484, E3 +68747.638}
SPL {X  -160.000, Y  +398.391, Z    +0.000, E1   +14.502, E3 +68766.464}
SPL {X  -160.000, Y  +395.999, Z    +0.000, E1   +14.484, E3 +68786.254}
SPL {X  -160.000, Y  +393.685, Z    +0.000, E1   +14.486, E3 +68805.326}
SPL {X  -159.999, Y  +391.313, Z    +0.000, E1   +14.479, E3 +68824.908}
SPL {X  -159.970, Y  +388.900, Z    +0.000, E1   +14.480, E3 +68844.793}
SPL {X  -159.903, Y  +386.417, Z    +0.000, E1   +14.475, E3 +68865.298}
SPL {X  -159.796, Y  +383.921, Z    +0.000, E1   +14.466, E3 +68885.953}
SPL {X  -159.651, Y  +381.443, Z    +0.000, E1   +14.453, E3 +68906.501}
SPL {X  -159.474, Y  +379.042, Z    +0.000, E1   +14.434, E3 +68926.465}
SPL {X  -159.316, Y  +377.219, Z    +0.000, E1   +14.400, E3 +68941.693}
ENDSPLINE

SPLINE
SPL {X  -159.452, Y  +378.767, Z    +0.000, E1   +11.887, E3 +68962.683}
SPL {X  -159.840, Y  +384.856, Z    +0.000, E1    +7.126, E3 +68981.654}
SPL {X  -159.991, Y  +390.336, Z    +0.000, E1    +2.803, E3 +68995.477}
SPL {X  -160.000, Y  +403.532, Z    +0.000, E1    -6.523, E3 +69013.198}
SPL {X  -160.000, Y  +409.023, Z    +0.000, E1   -10.003, E3 +69023.971}
SPL {X  -160.000, Y  +418.032, Z    +0.000, E1   -14.569, E3 +69048.830}
SPL {X  -160.000, Y  +420.561, Z    +0.000, E1   -14.816, E3 +69066.311}
SPL {X  -160.000, Y  +422.801, Z    +0.000, E1   -14.823, E3 +69084.259}
SPL {X  -160.000, Y  +425.518, Z    +0.000, E1   -14.845, E3 +69106.034}
SPL {X  -160.000, Y  +428.688, Z    +0.000, E1   -14.854, E3 +69131.442}
SPL {X  -160.000, Y  +431.971, Z    +0.000, E1   -14.849, E3 +69157.910}
SPL {X  -160.000, Y  +435.345, Z    +0.000, E1   -14.857, E3 +69184.961}
SPL {X  -160.000, Y  +438.732, Z    +0.000, E1   -14.858, E3 +69212.109}
SPL {X  -160.000, Y  +441.925, Z    +0.000, E1   -14.848, E3 +69237.779}
SPL {X  -160.000, Y  +444.299, Z    +0.000, E1   -14.809, E3 +69256.964}
SPL {X  -160.000, Y  +446.229, Z    +0.000, E1   -14.820, E3 +69272.383}
SPL {X  -160.000, Y  +448.987, Z    +0.000, E1   -14.868, E3 +69294.320}
SPL {X  -160.000, Y  +452.351, Z    +0.000, E1   -14.871, E3 +69321.296}
SPL {X  -160.000, Y  +455.709, Z    +0.000, E1   -14.880, E3 +69348.110}
SPL {X  -160.000, Y  +458.189, Z    +0.000, E1   -14.832, E3 +69368.111}
SPL {X  -160.000, Y  +459.885, Z    +0.000, E1   -14.825, E3 +69381.782}
SPL {X  -160.000, Y  +462.438, Z    +0.000, E1   -14.868, E3 +69402.192}
SPL {X  -160.000, Y  +465.575, Z    +0.000, E1   -14.849, E3 +69427.500}
SPL {X  -160.000, Y  +468.581, Z    +0.000, E1   -14.841, E3 +69451.733}
SPL {X  -160.000, Y  +471.795, Z    +0.000, E1   -14.854, E3 +69477.520}
SPL {X  -160.000, Y  +475.138, Z    +0.000, E1   -14.853, E3 +69504.371}
SPL {X  -160.000, Y  +477.981, Z    +0.000, E1   -14.823, E3 +69527.291}
SPL {X  -160.000, Y  +480.658, Z    +0.000, E1   -14.835, E3 +69548.767}
SPL {X  -160.000, Y  +483.534, Z    +0.000, E1   -14.838, E3 +69571.862}
SPL {X  -160.000, Y  +486.226, Z    +0.000, E1   -14.823, E3 +69593.527}
SPL {X  -160.000, Y  +488.751, Z    +0.000, E1   -14.827, E3 +69613.799}
SPL {X  -160.000, Y  +491.612, Z    +0.000, E1   -14.844, E3 +69636.722}
SPL {X  -160.000, Y  +494.417, Z    +0.000, E1   -14.827, E3 +69659.313}
SPL {X  -160.000, Y  +496.961, Z    +0.000, E1   -14.824, E3 +69679.757}
SPL {X  -160.000, Y  +499.610, Z    +0.000, E1   -14.830, E3 +69701.029}
SPL {X  -160.000, Y  +502.268, Z    +0.000, E1   -14.832, E3 +69722.298}
SPL {X  -160.000, Y  +505.041, Z    +0.000, E1   -14.849, E3 +69744.461}
SPL {X  -160.000, Y  +507.743, Z    +0.000, E1   -14.842, E3 +69766.085}
SPL {X  -160.000, Y  +510.437, Z    +0.000, E1   -14.860, E3 +69787.599}
SPL {X  -160.000, Y  +513.179, Z    +0.000, E1   -14.849, E3 +69809.646}
SPL {X  -160.000, Y  +515.613, Z    +0.000, E1   -14.829, E3 +69829.316}
SPL {X  -160.000, Y  +518.188, Z    +0.000, E1   -14.845, E3 +69849.946}
SPL {X  -160.000, Y  +520.790, Z    +0.000, E1   -14.839, E3 +69870.775}
SPL {X  -160.000, Y  +523.469, Z    +0.000, E1   -14.855, E3 +69892.223}
SPL {X  -160.000, Y  +526.403, Z    +0.000, E1   -14.858, E3 +69915.759}
SPL {X  -160.000, Y  +529.266, Z    +0.000, E1   -14.848, E3 +69938.767}
SPL {X  -160.000, Y  +531.688, Z    +0.000, E1   -14.826, E3 +69958.316}
SPL {X  -160.000, Y  +534.214, Z    +0.000, E1   -14.841, E3 +69978.579}
SPL {X  -160.000, Y  +537.002, Z    +0.000, E1   -14.839, E3 +70000.997}
SPL {X  -160.000, Y  +539.729, Z    +0.000, E1   -14.840, E3 +70022.809}
SPL {X  -160.000, Y  +542.408, Z    +0.000, E1   -14.839, E3 +70044.362}
SPL {X  -160.000, Y  +545.014, Z    +0.000, E1   -14.831, E3 +70065.307}
SPL {X  -160.000, Y  +547.659, Z    +0.000, E1   -14.839, E3 +70086.522}
SPL {X  -160.000, Y  +550.215, Z    +0.000, E1   -14.827, E3 +70107.087}
SPL {X  -160.000, Y  +552.762, Z    +0.000, E1   -14.836, E3 +70127.505}
SPL {X  -160.000, Y  +555.331, Z    +0.000, E1   -14.837, E3 +70148.046}
SPL {X  -160.000, Y  +558.235, Z    +0.000, E1   -14.869, E3 +70171.210}
SPL {X  -160.000, Y  +561.088, Z    +0.000, E1   -14.848, E3 +70194.128}
SPL {X  -160.000, Y  +563.693, Z    +0.000, E1   -14.852, E3 +70214.989}
SPL {X  -160.000, Y  +566.560, Z    +0.000, E1   -14.865, E3 +70237.966}
SPL {X  -160.000, Y  +569.305, Z    +0.000, E1   -14.848, E3 +70259.995}
SPL {X  -160.000, Y  +571.769, Z    +0.000, E1   -14.852, E3 +70279.740}
SPL {X  -160.000, Y  +574.366, Z    +0.000, E1   -14.855, E3 +70300.527}
SPL {X  -160.000, Y  +577.037, Z    +0.000, E1   -14.859, E3 +70321.927}
SPL {X  -160.000, Y  +579.855, Z    +0.000, E1   -14.869, E3 +70344.454}
SPL {X  -160.000, Y  +582.456, Z    +0.000, E1   -14.854, E3 +70365.314}
SPL {X  -160.000, Y  +585.083, Z    +0.000, E1   -14.866, E3 +70386.364}
SPL {X  -160.000, Y  +587.675, Z    +0.000, E1   -14.853, E3 +70407.155}
SPL {X  -160.000, Y  +590.216, Z    +0.000, E1   -14.864, E3 +70427.474}
SPL {X  -160.000, Y  +592.848, Z    +0.000, E1   -14.865, E3 +70448.525}
SPL {X  -160.000, Y  +595.342, Z    +0.000, E1   -14.848, E3 +70468.703}
SPL {X  -160.000, Y  +597.995, Z    +0.000, E1   -14.848, E3 +70490.043}
SPL {X  -160.000, Y  +600.731, Z    +0.000, E1   -14.846, E3 +70511.994}
SPL {X  -160.000, Y  +603.404, Z    +0.000, E1   -14.846, E3 +70533.430}
SPL {X  -160.000, Y  +605.923, Z    +0.000, E1   -14.838, E3 +70553.671}
SPL {X  -160.000, Y  +608.492, Z    +0.000, E1   -14.846, E3 +70574.275}
SPL {X  -160.000, Y  +611.345, Z    +0.000, E1   -14.856, E3 +70597.133}
SPL {X  -160.000, Y  +614.087, Z    +0.000, E1   -14.839, E3 +70619.192}
SPL {X  -160.000, Y  +616.566, Z    +0.000, E1   -14.839, E3 +70639.086}
SPL {X  -160.000, Y  +619.350, Z    +0.000, E1   -14.855, E3 +70661.374}
SPL {X  -160.000, Y  +622.198, Z    +0.000, E1   -14.846, E3 +70684.258}
SPL {X  -160.000, Y  +624.642, Z    +0.000, E1   -14.829, E3 +70703.931}
SPL {X  -160.000, Y  +627.119, Z    +0.000, E1   -14.843, E3 +70723.771}
SPL {X  -160.000, Y  +629.682, Z    +0.000, E1   -14.838, E3 +70744.340}
SPL {X  -160.000, Y  +632.223, Z    +0.000, E1   -14.841, E3 +70764.731}
SPL {X  -160.000, Y  +634.941, Z    +0.000, E1   -14.846, E3 +70786.529}
SPL {X  -160.000, Y  +637.723, Z    +0.000, E1   -14.844, E3 +70808.873}
SPL {X  -160.000, Y  +640.315, Z    +0.000, E1   -14.836, E3 +70829.670}
SPL {X  -160.000, Y  +643.085, Z    +0.000, E1   -14.865, E3 +70851.722}
SPL {X  -160.000, Y  +645.845, Z    +0.000, E1   -14.848, E3 +70873.910}
SPL {X  -160.000, Y  +648.229, Z    +0.000, E1   -14.834, E3 +70893.120}
SPL {X  -160.000, Y  +650.656, Z    +0.000, E1   -14.835, E3 +70912.676}
SPL {X  -160.000, Y  +653.134, Z    +0.000, E1   -14.827, E3 +70932.603}
SPL {X  -160.000, Y  +655.670, Z    +0.000, E1   -14.841, E3 +70952.897}
SPL {X  -160.000, Y  +658.349, Z    +0.000, E1   -14.842, E3 +70974.373}
SPL {X  -160.000, Y  +660.936, Z    +0.000, E1   -14.838, E3 +70995.125}
SPL {X  -160.000, Y  +663.567, Z    +0.000, E1   -14.845, E3 +71016.255}
SPL {X  -160.000, Y  +666.216, Z    +0.000, E1   -14.832, E3 +71037.572}
SPL {X  -159.997, Y  +668.731, Z    +0.000, E1   -14.834, E3 +71057.764}
SPL {X  -159.962, Y  +671.176, Z    +0.000, E1   -14.822, E3 +71077.475}
SPL {X  -159.895, Y  +673.507, Z    +0.000, E1   -14.821, E3 +71096.206}
SPL {X  -159.785, Y  +675.985, Z    +0.000, E1   -14.818, E3 +71116.208}
SPL {X  -159.627, Y  +678.622, Z    +0.000, E1   -14.804, E3 +71137.560}
SPL {X  -159.438, Y  +681.094, Z    +0.000, E1   -14.770, E3 +71157.732}
SPL {X  -159.262, Y  +683.054, Z    +0.000, E1   -14.719, E3 +71173.960}
ENDSPLINE

SPLINE
SPL {X  -159.661, Y  +678.114, Z    +0.000, E1    -9.575, E3 +71203.552}
SPL {X  -159.942, Y  +672.020, Z    +0.000, E1    -4.692, E3 +71222.179}
SPL {X  -160.000, Y  +664.971, Z    +0.000, E1    +0.516, E3 +71241.729}
SPL {X  -160.000, Y  +660.032, Z    +0.000, E1    +3.995, E3 +71253.672}
SPL {X  -160.000, Y  +652.280, Z    +0.000, E1    +8.913, E3 +71272.187}
SPL {X  -160.000, Y  +644.147, Z    +0.000, E1   +13.158, E3 +71295.738}
SPL {X  -160.000, Y  +641.594, Z    +0.000, E1   +13.488, E3 +71314.179}
SPL {X  -160.000, Y  +639.799, Z    +0.000, E1   +13.486, E3 +71330.089}
SPL {X  -160.000, Y  +637.896, Z    +0.000, E1   +13.493, E3 +71346.904}
SPL {X  -160.000, Y  +635.832, Z    +0.000, E1   +13.499, E3 +71365.162}
SPL {X  -160.000, Y  +633.839, Z    +0.000, E1   +13.489, E3 +71382.851}
SPL {X  -160.000, Y  +631.625, Z    +0.000, E1   +13.508, E3 +71402.392}
SPL {X  -160.000, Y  +629.417, Z    +0.000, E1   +13.491, E3 +71422.003}
SPL {X  -160.000, Y  +627.180, Z    +0.000, E1   +13.508, E3 +71441.757}
SPL {X  -160.000, Y  +624.970, Z    +0.000, E1   +13.490, E3 +71461.408}
SPL {X  -160.000, Y  +623.020, Z    +0.000, E1   +13.491, E3 +71478.637}
SPL {X  -160.000, Y  +620.888, Z    +0.000, E1   +13.501, E3 +71497.500}
SPL {X  -160.000, Y  +618.790, Z    +0.000, E1   +13.488, E3 +71516.122}
SPL {X  -160.000, Y  +616.631, Z    +0.000, E1   +13.504, E3 +71535.176}
SPL {X  -160.000, Y  +614.230, Z    +0.000, E1   +13.510, E3 +71556.372}
SPL {X  -160.000, Y  +612.132, Z    +0.000, E1   +13.485, E3 +71575.088}
SPL {X  -160.000, Y  +610.405, Z    +0.000, E1   +13.477, E3 +71590.461}
SPL {X  -160.000, Y  +608.437, Z    +0.000, E1   +13.502, E3 +71607.717}
SPL {X  -160.000, Y  +606.281, Z    +0.000, E1   +13.502, E3 +71626.734}
SPL {X  -160.000, Y  +604.124, Z    +0.000, E1   +13.513, E3 +71645.789}
SPL {X  -160.000, Y  +601.878, Z    +0.000, E1   +13.505, E3 +71665.687}
SPL {X  -160.000, Y  +599.648, Z    +0.000, E1   +13.506, E3 +71685.463}
SPL {X  -160.000, Y  +597.673, Z    +0.000, E1   +13.479, E3 +71703.137}
SPL {X  -160.000, Y  +595.601, Z    +0.000, E1   +13.499, E3 +71721.420}
SPL {X  -160.000, Y  +593.187, Z    +0.000, E1   +13.500, E3 +71742.800}
SPL {X  -160.000, Y  +591.079, Z    +0.000, E1   +13.483, E3 +71761.526}
SPL {X  -160.000, Y  +589.151, Z    +0.000, E1   +13.489, E3 +71778.577}
SPL {X  -160.000, Y  +586.908, Z    +0.000, E1   +13.501, E3 +71798.423}
SPL {X  -160.000, Y  +584.660, Z    +0.000, E1   +13.490, E3 +71818.364}
SPL {X  -160.000, Y  +582.409, Z    +0.000, E1   +13.499, E3 +71838.283}
SPL {X  -160.000, Y  +580.150, Z    +0.000, E1   +13.490, E3 +71858.329}
SPL {X  -160.000, Y  +577.953, Z    +0.000, E1   +13.493, E3 +71877.788}
SPL {X  -160.000, Y  +575.630, Z    +0.000, E1   +13.502, E3 +71898.271}
SPL {X  -160.000, Y  +573.418, Z    +0.000, E1   +13.502, E3 +71917.779}
SPL {X  -160.000, Y  +571.226, Z    +0.000, E1   +13.520, E3 +71936.988}
SPL {X  -160.000, Y  +569.166, Z    +0.000, E1   +13.512, E3 +71955.179}
SPL {X  -160.000, Y  +567.275, Z    +0.000, E1   +13.517, E3 +71971.846}
SPL {X  -160.000, Y  +565.259, Z    +0.000, E1   +13.523, E3 +71989.635}
SPL {X  -160.000, Y  +563.305, Z    +0.000, E1   +13.512, E3 +72006.973}
SPL {X  -160.000, Y  +561.240, Z    +0.000, E1   +13.521, E3 +72025.235}
SPL {X  -160.000, Y  +558.881, Z    +0.000, E1   +13.524, E3 +72046.077}
SPL {X  -160.000, Y  +556.697, Z    +0.000, E1   +13.510, E3 +72065.463}
SPL {X  -160.000, Y  +554.624, Z    +0.000, E1   +13.512, E3 +72083.794}
SPL {X  -160.000, Y  +552.465, Z    +0.000, E1   +13.514, E3 +72102.878}
SPL {X  -160.000, Y  +550.315, Z    +0.000, E1   +13.514, E3 +72121.872}
SPL {X  -160.000, Y  +548.056, Z    +0.000, E1   +13.519, E3 +72141.873}
SPL {X  -160.000, Y  +545.826, Z    +0.000, E1   +13.501, E3 +72161.751}
SPL {X  -160.000, Y  +543.677, Z    +0.000, E1   +13.502, E3 +72180.809}
SPL {X  -160.000, Y  +541.664, Z    +0.000, E1   +13.489, E3 +72198.694}
SPL {X  -160.000, Y  +539.659, Z    +0.000, E1   +13.494, E3 +72216.454}
SPL {X  -160.000, Y  +537.370, Z    +0.000, E1   +13.501, E3 +72236.693}
SPL {X  -160.000, Y  +535.056, Z    +0.000, E1   +13.506, E3 +72257.089}
SPL {X  -160.000, Y  +532.975, Z    +0.000, E1   +13.494, E3 +72275.576}
SPL {X  -160.000, Y  +530.925, Z    +0.000, E1   +13.499, E3 +72293.737}
SPL {X  -160.000, Y  +528.768, Z    +0.000, E1   +13.498, E3 +72312.839}
SPL {X  -160.000, Y  +526.547, Z    +0.000, E1   +13.499, E3 +72332.507}
SPL {X  -160.000, Y  +523.964, Z    +0.000, E1   +13.742, E3 +72352.012}
SPL {X  -160.000, Y  +513.971, Z    +0.000, E1   +18.644, E3 +72370.924}
SPL {X  -160.000, Y  +513.562, Z    +0.000, E1   +16.972, E3 +72390.801}
SPL {X  -160.000, Y  +513.358, Z    +0.000, E1   +15.267, E3 +72411.072}
SPL {X  -160.000, Y  +512.244, Z    +0.000, E1   +14.473, E3 +72429.529}
SPL {X  -160.000, Y  +509.675, Z    +0.000, E1   +14.481, E3 +72450.672}
SPL {X  -160.000, Y  +507.162, Z    +0.000, E1   +14.470, E3 +72471.412}
SPL {X  -160.000, Y  +504.735, Z    +0.000, E1   +14.473, E3 +72491.384}
SPL {X  -160.000, Y  +502.261, Z    +0.000, E1   +14.476, E3 +72511.720}
SPL {X  -160.000, Y  +499.798, Z    +0.000, E1   +14.482, E3 +72531.922}
SPL {X  -160.000, Y  +497.435, Z    +0.000, E1   +14.476, E3 +72551.399}
SPL {X  -160.000, Y  +495.089, Z    +0.000, E1   +14.475, E3 +72570.765}
SPL {X  -160.000, Y  +492.764, Z    +0.000, E1   +14.469, E3 +72589.937}
SPL {X  -160.000, Y  +490.292, Z    +0.000, E1   +14.476, E3 +72610.338}
SPL {X  -160.000, Y  +487.641, Z    +0.000, E1   +14.470, E3 +72632.234}
SPL {X  -160.000, Y  +485.054, Z    +0.000, E1   +14.460, E3 +72653.677}
SPL {X  -160.000, Y  +482.421, Z    +0.000, E1   +14.461, E3 +72675.395}
SPL {X  -160.000, Y  +480.000, Z    +0.000, E1   +14.451, E3 +72695.359}
SPL {X  -160.000, Y  +477.551, Z    +0.000, E1   +14.466, E3 +72715.488}
SPL {X  -160.000, Y  +475.253, Z    +0.000, E1   +14.450, E3 +72734.462}
SPL {X  -160.000, Y  +473.070, Z    +0.000, E1   +14.454, E3 +72752.483}
SPL {X  -160.000, Y  +470.603, Z    +0.000, E1   +14.464, E3 +72772.783}
SPL {X  -160.000, Y  +468.243, Z    +0.000, E1   +14.458, E3 +72792.182}
SPL {X  -160.000, Y  +465.791, Z    +0.000, E1   +14.475, E3 +72812.326}
SPL {X  -160.000, Y  +463.103, Z    +0.000, E1   +14.474, E3 +72834.475}
SPL {X  -160.000, Y  +460.743, Z    +0.000, E1   +14.465, E3 +72853.883}
SPL {X  -160.000, Y  +458.292, Z    +0.000, E1   +14.492, E3 +72873.883}
SPL {X  -160.000, Y  +455.874, Z    +0.000, E1   +14.484, E3 +72893.740}
SPL {X  -160.000, Y  +453.555, Z    +0.000, E1   +14.488, E3 +72912.820}
SPL {X  -160.000, Y  +451.093, Z    +0.000, E1   +14.485, E3 +72933.132}
SPL {X  -160.000, Y  +448.700, Z    +0.000, E1   +14.483, E3 +72952.821}
SPL {X  -160.000, Y  +446.277, Z    +0.000, E1   +14.485, E3 +72972.745}
SPL {X  -160.000, Y  +443.879, Z    +0.000, E1   +14.485, E3 +72992.483}
SPL {X  -160.000, Y  +441.447, Z    +0.000, E1   +14.485, E3 +73012.490}
SPL {X  -160.000, Y  +439.006, Z    +0.000, E1   +14.488, E3 +73032.573}
SPL {X  -160.000, Y  +436.311, Z    +0.000, E1   +14.498, E3 +73054.732}
SPL {X  -160.000, Y  +433.559, Z    +0.000, E1   +14.491, E3 +73077.401}
SPL {X  -160.000, Y  +431.162, Z    +0.000, E1   +14.479, E3 +73097.153}
SPL {X  -160.000, Y  +429.152, Z    +0.000, E1   +14.469, E3 +73113.734}
SPL {X  -160.000, Y  +426.863, Z    +0.000, E1   +14.490, E3 +73132.513}
SPL {X  -160.000, Y  +424.653, Z    +0.000, E1   +14.467, E3 +73150.772}
SPL {X  -160.000, Y  +422.337, Z    +0.000, E1   +14.492, E3 +73169.757}
SPL {X  -160.000, Y  +419.639, Z    +0.000, E1   +14.504, E3 +73191.797}
SPL {X  -160.000, Y  +417.127, Z    +0.000, E1   +14.501, E3 +73212.388}
SPL {X  -160.000, Y  +414.849, Z    +0.000, E1   +14.496, E3 +73231.122}
SPL {X  -160.000, Y  +412.396, Z    +0.000, E1   +14.505, E3 +73251.311}
SPL {X  -160.000, Y  +409.815, Z    +0.000, E1   +14.498, E3 +73272.565}
SPL {X  -160.000, Y  +407.614, Z    +0.000, E1   +14.484, E3 +73290.690}
SPL {X  -160.000, Y  +405.406, Z    +0.000, E1   +14.501, E3 +73308.753}
SPL {X  -160.000, Y  +402.958, Z    +0.000, E1   +14.500, E3 +73328.923}
SPL {X  -160.000, Y  +400.690, Z    +0.000, E1   +14.484, E3 +73347.635}
SPL {X  -160.000, Y  +398.391, Z    +0.000, E1   +14.502, E3 +73366.461}
SPL {X  -160.000, Y  +395.999, Z    +0.000, E1   +14.484, E3 +73386.251}
SPL {X  -160.000, Y  +393.685, Z    +0.000, E1   +14.486, E3 +73405.323}
SPL {X  -159.999, Y  +391.313, Z    +0.000, E1   +14.479, E3 +73424.905}
SPL {X  -159.970, Y  +388.900, Z    +0.000, E1   +14.480, E3 +73444.789}
SPL {X  -159.903, Y  +386.417, Z    +0.000, E1   +14.475, E3 +73465.295}
SPL {X  -159.796, Y  +383.921, Z    +0.000, E1   +14.466, E3 +73485.950}
SPL {X  -159.651, Y  +381.443, Z    +0.000, E1   +14.453, E3 +73506.498}
SPL {X  -159.474, Y  +379.042, Z    +0.000, E1   +14.434, E3 +73526.462}
SPL {X  -159.316, Y  +377.219, Z    +0.000, E1   +14.400, E3 +73541.690}
ENDSPLINE

SPLINE
SPL {X  -159.452, Y  +378.767, Z    +0.000, E1   +11.887, E3 +73562.679}
SPL {X  -159.840, Y  +384.856, Z    +0.000, E1    +7.126, E3 +73581.651}
SPL {X  -159.991, Y  +390.336, Z    +0.000, E1    +2.803, E3 +73595.474}
SPL {X  -160.000, Y  +403.532, Z    +0.000, E1    -6.523, E3 +73613.194}
SPL {X  -160.000, Y  +409.023, Z    +0.000, E1   -10.003, E3 +73623.968}
SPL {X  -160.000, Y  +418.032, Z    +0.000, E1   -14.569, E3 +73648.827}
SPL {X  -160.000, Y  +420.561, Z    +0.000, E1   -14.816, E3 +73666.307}
SPL {X  -160.000, Y  +422.801, Z    +0.000, E1   -14.823, E3 +73684.256}
SPL {X  -160.000, Y  +425.518, Z    +0.000, E1   -14.845, E3 +73706.030}
SPL {X  -160.000, Y  +428.688, Z    +0.000, E1   -14.854, E3 +73731.439}
SPL {X  -160.000, Y  +431.971, Z    +0.000, E1   -14.849, E3 +73757.907}
SPL {X  -160.000, Y  +435.345, Z    +0.000, E1   -14.857, E3 +73784.957}
SPL {X  -160.000, Y  +438.732, Z    +0.000, E1   -14.858, E3 +73812.106}
SPL {X  -160.000, Y  +441.925, Z    +0.000, E1   -14.848, E3 +73837.776}
SPL {X  -160.000, Y  +444.299, Z    +0.000, E1   -14.809, E3 +73856.961}
SPL {X  -160.000, Y  +446.229, Z    +0.000, E1   -14.820, E3 +73872.380}
SPL {X  -160.000, Y  +448.987, Z    +0.000, E1   -14.868, E3 +73894.316}
SPL {X  -160.000, Y  +452.351, Z    +0.000, E1   -14.871, E3 +73921.292}
SPL {X  -160.000, Y  +455.709, Z    +0.000, E1   -14.880, E3 +73948.107}
SPL {X  -160.000, Y  +458.189, Z    +0.000, E1   -14.832, E3 +73968.108}
SPL {X  -160.000, Y  +459.885, Z    +0.000, E1   -14.825, E3 +73981.779}
SPL {X  -160.000, Y  +462.438, Z    +0.000, E1   -14.868, E3 +74002.189}
SPL {X  -160.000, Y  +465.575, Z    +0.000, E1   -14.849, E3 +74027.497}
SPL {X  -160.000, Y  +468.581, Z    +0.000, E1   -14.841, E3 +74051.729}
SPL {X  -160.000, Y  +471.795, Z    +0.000, E1   -14.854, E3 +74077.517}
SPL {X  -160.000, Y  +475.138, Z    +0.000, E1   -14.853, E3 +74104.367}
SPL {X  -160.000, Y  +477.981, Z    +0.000, E1   -14.823, E3 +74127.288}
SPL {X  -160.000, Y  +480.658, Z    +0.000, E1   -14.835, E3 +74148.764}
SPL {X  -160.000, Y  +483.534, Z    +0.000, E1   -14.838, E3 +74171.858}
SPL {X  -160.000, Y  +486.226, Z    +0.000, E1   -14.823, E3 +74193.524}
SPL {X  -160.000, Y  +488.751, Z    +0.000, E1   -14.827, E3 +74213.796}
SPL {X  -160.000, Y  +491.612, Z    +0.000, E1   -14.844, E3 +74236.719}
SPL {X  -160.000, Y  +494.417, Z    +0.000, E1   -14.827, E3 +74259.309}
SPL {X  -160.000, Y  +496.961, Z    +0.000, E1   -14.824, E3 +74279.753}
SPL {X  -160.000, Y  +499.610, Z    +0.000, E1   -14.830, E3 +74301.026}
SPL {X  -160.000, Y  +502.268, Z    +0.000, E1   -14.832, E3 +74322.295}
SPL {X  -160.000, Y  +505.041, Z    +0.000, E1   -14.849, E3 +74344.458}
SPL {X  -160.000, Y  +507.743, Z    +0.000, E1   -14.842, E3 +74366.082}
SPL {X  -160.000, Y  +510.437, Z    +0.000, E1   -14.860, E3 +74387.595}
SPL {X  -160.000, Y  +513.179, Z    +0.000, E1   -14.849, E3 +74409.643}
SPL {X  -160.000, Y  +515.613, Z    +0.000, E1   -14.829, E3 +74429.313}
SPL {X  -160.000, Y  +518.188, Z    +0.000, E1   -14.845, E3 +74449.943}
SPL {X  -160.000, Y  +520.790, Z    +0.000, E1   -14.839, E3 +74470.771}
SPL {X  -160.000, Y  +523.469, Z    +0.000, E1   -14.855, E3 +74492.220}
SPL {X  -160.000, Y  +526.403, Z    +0.000, E1   -14.858, E3 +74515.756}
SPL {X  -160.000, Y  +529.266, Z    +0.000, E1   -14.848, E3 +74538.763}
SPL {X  -160.000, Y  +531.688, Z    +0.000, E1   -14.826, E3 +74558.313}
SPL {X  -160.000, Y  +534.214, Z    +0.000, E1   -14.841, E3 +74578.576}
SPL {X  -160.000, Y  +537.002, Z    +0.000, E1   -14.839, E3 +74600.994}
SPL {X  -160.000, Y  +539.729, Z    +0.000, E1   -14.840, E3 +74622.806}
SPL {X  -160.000, Y  +542.408, Z    +0.000, E1   -14.839, E3 +74644.359}
SPL {X  -160.000, Y  +545.014, Z    +0.000, E1   -14.831, E3 +74665.304}
SPL {X  -160.000, Y  +547.659, Z    +0.000, E1   -14.839, E3 +74686.519}
SPL {X  -160.000, Y  +550.215, Z    +0.000, E1   -14.827, E3 +74707.084}
SPL {X  -160.000, Y  +552.762, Z    +0.000, E1   -14.836, E3 +74727.502}
SPL {X  -160.000, Y  +555.331, Z    +0.000, E1   -14.837, E3 +74748.043}
SPL {X  -160.000, Y  +558.235, Z    +0.000, E1   -14.869, E3 +74771.206}
SPL {X  -160.000, Y  +561.088, Z    +0.000, E1   -14.848, E3 +74794.125}
SPL {X  -160.000, Y  +563.693, Z    +0.000, E1   -14.852, E3 +74814.985}
SPL {X  -160.000, Y  +566.560, Z    +0.000, E1   -14.865, E3 +74837.963}
SPL {X  -160.000, Y  +569.305, Z    +0.000, E1   -14.848, E3 +74859.991}
SPL {X  -160.000, Y  +571.769, Z    +0.000, E1   -14.852, E3 +74879.737}
SPL {X  -160.000, Y  +574.366, Z    +0.000, E1   -14.855, E3 +74900.524}
SPL {X  -160.000, Y  +577.037, Z    +0.000, E1   -14.859, E3 +74921.924}
SPL {X  -160.000, Y  +579.855, Z    +0.000, E1   -14.869, E3 +74944.451}
SPL {X  -160.000, Y  +582.456, Z    +0.000, E1   -14.854, E3 +74965.311}
SPL {X  -160.000, Y  +585.083, Z    +0.000, E1   -14.866, E3 +74986.361}
SPL {X  -160.000, Y  +587.675, Z    +0.000, E1   -14.853, E3 +75007.152}
SPL {X  -160.000, Y  +590.216, Z    +0.000, E1   -14.864, E3 +75027.471}
SPL {X  -160.000, Y  +592.848, Z    +0.000, E1   -14.865, E3 +75048.522}
SPL {X  -160.000, Y  +595.342, Z    +0.000, E1   -14.848, E3 +75068.700}
SPL {X  -160.000, Y  +597.995, Z    +0.000, E1   -14.848, E3 +75090.039}
SPL {X  -160.000, Y  +600.731, Z    +0.000, E1   -14.846, E3 +75111.991}
SPL {X  -160.000, Y  +603.404, Z    +0.000, E1   -14.846, E3 +75133.427}
SPL {X  -160.000, Y  +605.923, Z    +0.000, E1   -14.838, E3 +75153.668}
SPL {X  -160.000, Y  +608.492, Z    +0.000, E1   -14.846, E3 +75174.271}
SPL {X  -160.000, Y  +611.345, Z    +0.000, E1   -14.856, E3 +75197.130}
SPL {X  -160.000, Y  +614.087, Z    +0.000, E1   -14.839, E3 +75219.189}
SPL {X  -160.000, Y  +616.566, Z    +0.000, E1   -14.839, E3 +75239.083}
SPL {X  -160.000, Y  +619.350, Z    +0.000, E1   -14.855, E3 +75261.371}
SPL {X  -160.000, Y  +622.198, Z    +0.000, E1   -14.846, E3 +75284.255}
SPL {X  -160.000, Y  +624.642, Z    +0.000, E1   -14.829, E3 +75303.928}
SPL {X  -160.000, Y  +627.119, Z    +0.000, E1   -14.843, E3 +75323.768}
SPL {X  -160.000, Y  +629.682, Z    +0.000, E1   -14.838, E3 +75344.337}
SPL {X  -160.000, Y  +632.223, Z    +0.000, E1   -14.841, E3 +75364.728}
SPL {X  -160.000, Y  +634.941, Z    +0.000, E1   -14.846, E3 +75386.525}
SPL {X  -160.000, Y  +637.723, Z    +0.000, E1   -14.844, E3 +75408.870}
SPL {X  -160.000, Y  +640.315, Z    +0.000, E1   -14.836, E3 +75429.667}
SPL {X  -160.000, Y  +643.085, Z    +0.000, E1   -14.865, E3 +75451.719}
SPL {X  -160.000, Y  +645.845, Z    +0.000, E1   -14.848, E3 +75473.907}
SPL {X  -160.000, Y  +648.229, Z    +0.000, E1   -14.834, E3 +75493.117}
SPL {X  -160.000, Y  +650.656, Z    +0.000, E1   -14.835, E3 +75512.673}
SPL {X  -160.000, Y  +653.134, Z    +0.000, E1   -14.827, E3 +75532.600}
SPL {X  -160.000, Y  +655.670, Z    +0.000, E1   -14.841, E3 +75552.894}
SPL {X  -160.000, Y  +658.349, Z    +0.000, E1   -14.842, E3 +75574.370}
SPL {X  -160.000, Y  +660.936, Z    +0.000, E1   -14.838, E3 +75595.122}
SPL {X  -160.000, Y  +663.567, Z    +0.000, E1   -14.845, E3 +75616.252}
SPL {X  -160.000, Y  +666.216, Z    +0.000, E1   -14.832, E3 +75637.568}
SPL {X  -159.997, Y  +668.731, Z    +0.000, E1   -14.834, E3 +75657.760}
SPL {X  -159.962, Y  +671.176, Z    +0.000, E1   -14.822, E3 +75677.472}
SPL {X  -159.895, Y  +673.507, Z    +0.000, E1   -14.821, E3 +75696.203}
SPL {X  -159.785, Y  +675.985, Z    +0.000, E1   -14.818, E3 +75716.204}
SPL {X  -159.627, Y  +678.622, Z    +0.000, E1   -14.804, E3 +75737.557}
SPL {X  -159.438, Y  +681.094, Z    +0.000, E1   -14.770, E3 +75757.729}
SPL {X  -159.262, Y  +683.054, Z    +0.000, E1   -14.719, E3 +75773.957}
ENDSPLINE

SPLINE
SPL {X  -159.661, Y  +678.114, Z    +0.000, E1    -9.575, E3 +75803.549}
SPL {X  -159.942, Y  +672.020, Z    +0.000, E1    -4.692, E3 +75822.176}
SPL {X  -160.000, Y  +664.971, Z    +0.000, E1    +0.516, E3 +75841.726}
SPL {X  -160.000, Y  +660.032, Z    +0.000, E1    +3.995, E3 +75853.669}
SPL {X  -160.000, Y  +652.280, Z    +0.000, E1    +8.913, E3 +75872.184}
SPL {X  -160.000, Y  +644.147, Z    +0.000, E1   +13.158, E3 +75895.734}
SPL {X  -160.000, Y  +641.594, Z    +0.000, E1   +13.488, E3 +75914.175}
SPL {X  -160.000, Y  +639.799, Z    +0.000, E1   +13.486, E3 +75930.085}
SPL {X  -160.000, Y  +637.896, Z    +0.000, E1   +13.493, E3 +75946.900}
SPL {X  -160.000, Y  +635.832, Z    +0.000, E1   +13.499, E3 +75965.159}
SPL {X  -160.000, Y  +633.839, Z    +0.000, E1   +13.489, E3 +75982.848}
SPL {X  -160.000, Y  +631.625, Z    +0.000, E1   +13.508, E3 +76002.389}
SPL {X  -160.000, Y  +629.417, Z    +0.000, E1   +13.491, E3 +76022.000}
SPL {X  -160.000, Y  +627.180, Z    +0.000, E1   +13.508, E3 +76041.754}
SPL {X  -160.000, Y  +624.970, Z    +0.000, E1   +13.490, E3 +76061.404}
SPL {X  -160.000, Y  +623.020, Z    +0.000, E1   +13.491, E3 +76078.634}
SPL {X  -160.000, Y  +620.888, Z    +0.000, E1   +13.501, E3 +76097.496}
SPL {X  -160.000, Y  +618.790, Z    +0.000, E1   +13.488, E3 +76116.119}
SPL {X  -160.000, Y  +616.631, Z    +0.000, E1   +13.504, E3 +76135.172}
SPL {X  -160.000, Y  +614.230, Z    +0.000, E1   +13.510, E3 +76156.368}
SPL {X  -160.000, Y  +612.132, Z    +0.000, E1   +13.485, E3 +76175.085}
SPL {X  -160.000, Y  +610.405, Z    +0.000, E1   +13.477, E3 +76190.458}
SPL {X  -160.000, Y  +608.437, Z    +0.000, E1   +13.502, E3 +76207.713}
SPL {X  -160.000, Y  +606.281, Z    +0.000, E1   +13.502, E3 +76226.731}
SPL {X  -160.000, Y  +604.124, Z    +0.000, E1   +13.513, E3 +76245.786}
SPL {X  -160.000, Y  +601.878, Z    +0.000, E1   +13.505, E3 +76265.683}
SPL {X  -160.000, Y  +599.648, Z    +0.000, E1   +13.506, E3 +76285.460}
SPL {X  -160.000, Y  +597.673, Z    +0.000, E1   +13.479, E3 +76303.134}
SPL {X  -160.000, Y  +595.601, Z    +0.000, E1   +13.499, E3 +76321.417}
SPL {X  -160.000, Y  +593.187, Z    +0.000, E1   +13.500, E3 +76342.797}
SPL {X  -160.000, Y  +591.079, Z    +0.000, E1   +13.483, E3 +76361.523}
SPL {X  -160.000, Y  +589.151, Z    +0.000, E1   +13.489, E3 +76378.574}
SPL {X  -160.000, Y  +586.908, Z    +0.000, E1   +13.501, E3 +76398.420}
SPL {X  -160.000, Y  +584.660, Z    +0.000, E1   +13.490, E3 +76418.361}
SPL {X  -160.000, Y  +582.409, Z    +0.000, E1   +13.499, E3 +76438.279}
SPL {X  -160.000, Y  +580.150, Z    +0.000, E1   +13.490, E3 +76458.326}
SPL {X  -160.000, Y  +577.953, Z    +0.000, E1   +13.493, E3 +76477.784}
SPL {X  -160.000, Y  +575.630, Z    +0.000, E1   +13.502, E3 +76498.268}
SPL {X  -160.000, Y  +573.418, Z    +0.000, E1   +13.502, E3 +76517.776}
SPL {X  -160.000, Y  +571.226, Z    +0.000, E1   +13.520, E3 +76536.985}
SPL {X  -160.000, Y  +569.166, Z    +0.000, E1   +13.512, E3 +76555.175}
SPL {X  -160.000, Y  +567.275, Z    +0.000, E1   +13.517, E3 +76571.843}
SPL {X  -160.000, Y  +565.259, Z    +0.000, E1   +13.523, E3 +76589.632}
SPL {X  -160.000, Y  +563.305, Z    +0.000, E1   +13.512, E3 +76606.970}
SPL {X  -160.000, Y  +561.240, Z    +0.000, E1   +13.521, E3 +76625.232}
SPL {X  -160.000, Y  +558.881, Z    +0.000, E1   +13.524, E3 +76646.074}
SPL {X  -160.000, Y  +556.697, Z    +0.000, E1   +13.510, E3 +76665.460}
SPL {X  -160.000, Y  +554.624, Z    +0.000, E1   +13.512, E3 +76683.791}
SPL {X  -160.000, Y  +552.465, Z    +0.000, E1   +13.514, E3 +76702.875}
SPL {X  -160.000, Y  +550.315, Z    +0.000, E1   +13.514, E3 +76721.869}
SPL {X  -160.000, Y  +548.056, Z    +0.000, E1   +13.519, E3 +76741.870}
SPL {X  -160.000, Y  +545.826, Z    +0.000, E1   +13.501, E3 +76761.748}
SPL {X  -160.000, Y  +543.677, Z    +0.000, E1   +13.502, E3 +76780.806}
SPL {X  -160.000, Y  +541.664, Z    +0.000, E1   +13.489, E3 +76798.691}
SPL {X  -160.000, Y  +539.659, Z    +0.000, E1   +13.494, E3 +76816.451}
SPL {X  -160.000, Y  +537.370, Z    +0.000, E1   +13.501, E3 +76836.690}
SPL {X  -160.000, Y  +535.056, Z    +0.000, E1   +13.506, E3 +76857.086}
SPL {X  -160.000, Y  +532.975, Z    +0.000, E1   +13.494, E3 +76875.572}
SPL {X  -160.000, Y  +530.925, Z    +0.000, E1   +13.499, E3 +76893.734}
SPL {X  -160.000, Y  +528.768, Z    +0.000, E1   +13.498, E3 +76912.835}
SPL {X  -160.000, Y  +526.547, Z    +0.000, E1   +13.499, E3 +76932.504}
SPL {X  -160.000, Y  +523.964, Z    +0.000, E1   +13.742, E3 +76952.009}
SPL {X  -160.000, Y  +513.971, Z    +0.000, E1   +18.644, E3 +76970.921}
SPL {X  -160.000, Y  +513.562, Z    +0.000, E1   +16.972, E3 +76990.797}
SPL {X  -160.000, Y  +513.358, Z    +0.000, E1   +15.267, E3 +77011.069}
SPL {X  -160.000, Y  +512.244, Z    +0.000, E1   +14.473, E3 +77029.526}
SPL {X  -160.000, Y  +509.675, Z    +0.000, E1   +14.481, E3 +77050.669}
SPL {X  -160.000, Y  +507.162, Z    +0.000, E1   +14.470, E3 +77071.409}
SPL {X  -160.000, Y  +504.735, Z    +0.000, E1   +14.473, E3 +77091.380}
SPL {X  -160.000, Y  +502.261, Z    +0.000, E1   +14.476, E3 +77111.717}
SPL {X  -160.000, Y  +499.798, Z    +0.000, E1   +14.482, E3 +77131.919}
SPL {X  -160.000, Y  +497.435, Z    +0.000, E1   +14.476, E3 +77151.395}
SPL {X  -160.000, Y  +495.089, Z    +0.000, E1   +14.475, E3 +77170.762}
SPL {X  -160.000, Y  +492.764, Z    +0.000, E1   +14.469, E3 +77189.934}
SPL {X  -160.000, Y  +490.292, Z    +0.000, E1   +14.476, E3 +77210.335}
SPL {X  -160.000, Y  +487.641, Z    +0.000, E1   +14.470, E3 +77232.231}
SPL {X  -160.000, Y  +485.054, Z    +0.000, E1   +14.460, E3 +77253.673}
SPL {X  -160.000, Y  +482.421, Z    +0.000, E1   +14.461, E3 +77275.392}
SPL {X  -160.000, Y  +480.000, Z    +0.000, E1   +14.451, E3 +77295.356}
SPL {X  -160.000, Y  +477.551, Z    +0.000, E1   +14.466, E3 +77315.484}
SPL {X  -160.000, Y  +475.253, Z    +0.000, E1   +14.450, E3 +77334.459}
SPL {X  -160.000, Y  +473.070, Z    +0.000, E1   +14.454, E3 +77352.480}
SPL {X  -160.000, Y  +470.603, Z    +0.000, E1   +14.464, E3 +77372.780}
SPL {X  -160.000, Y  +468.243, Z    +0.000, E1   +14.458, E3 +77392.179}
SPL {X  -160.000, Y  +465.791, Z    +0.000, E1   +14.475, E3 +77412.323}
SPL {X  -160.000, Y  +463.103, Z    +0.000, E1   +14.474, E3 +77434.472}
SPL {X  -160.000, Y  +460.743, Z    +0.000, E1   +14.465, E3 +77453.880}
SPL {X  -160.000, Y  +458.292, Z    +0.000, E1   +14.492, E3 +77473.880}
SPL {X  -160.000, Y  +455.874, Z    +0.000, E1   +14.484, E3 +77493.737}
SPL {X  -160.000, Y  +453.555, Z    +0.000, E1   +14.488, E3 +77512.816}
SPL {X  -160.000, Y  +451.093, Z    +0.000, E1   +14.485, E3 +77533.128}
SPL {X  -160.000, Y  +448.700, Z    +0.000, E1   +14.483, E3 +77552.818}
SPL {X  -160.000, Y  +446.277, Z    +0.000, E1   +14.485, E3 +77572.742}
SPL {X  -160.000, Y  +443.879, Z    +0.000, E1   +14.485, E3 +77592.480}
SPL {X  -160.000, Y  +441.447, Z    +0.000, E1   +14.485, E3 +77612.487}
SPL {X  -160.000, Y  +439.006, Z    +0.000, E1   +14.488, E3 +77632.570}
SPL {X  -160.000, Y  +436.311, Z    +0.000, E1   +14.498, E3 +77654.729}
SPL {X  -160.000, Y  +433.559, Z    +0.000, E1   +14.491, E3 +77677.398}
SPL {X  -160.000, Y  +431.162, Z    +0.000, E1   +14.479, E3 +77697.150}
SPL {X  -160.000, Y  +429.152, Z    +0.000, E1   +14.469, E3 +77713.731}
SPL {X  -160.000, Y  +426.863, Z    +0.000, E1   +14.490, E3 +77732.510}
SPL {X  -160.000, Y  +424.653, Z    +0.000, E1   +14.467, E3 +77750.769}
SPL {X  -160.000, Y  +422.337, Z    +0.000, E1   +14.492, E3 +77769.753}
SPL {X  -160.000, Y  +419.639, Z    +0.000, E1   +14.504, E3 +77791.793}
SPL {X  -160.000, Y  +417.127, Z    +0.000, E1   +14.501, E3 +77812.385}
SPL {X  -160.000, Y  +414.849, Z    +0.000, E1   +14.496, E3 +77831.119}
SPL {X  -160.000, Y  +412.396, Z    +0.000, E1   +14.505, E3 +77851.308}
SPL {X  -160.000, Y  +409.815, Z    +0.000, E1   +14.498, E3 +77872.562}
SPL {X  -160.000, Y  +407.614, Z    +0.000, E1   +14.484, E3 +77890.687}
SPL {X  -160.000, Y  +405.406, Z    +0.000, E1   +14.501, E3 +77908.750}
SPL {X  -160.000, Y  +402.958, Z    +0.000, E1   +14.500, E3 +77928.920}
SPL {X  -160.000, Y  +400.690, Z    +0.000, E1   +14.484, E3 +77947.632}
SPL {X  -160.000, Y  +398.391, Z    +0.000, E1   +14.502, E3 +77966.458}
SPL {X  -160.000, Y  +395.999, Z    +0.000, E1   +14.484, E3 +77986.248}
SPL {X  -160.000, Y  +393.685, Z    +0.000, E1   +14.486, E3 +78005.320}
SPL {X  -159.999, Y  +391.313, Z    +0.000, E1   +14.479, E3 +78024.902}
SPL {X  -159.970, Y  +388.900, Z    +0.000, E1   +14.480, E3 +78044.786}
SPL {X  -159.903, Y  +386.417, Z    +0.000, E1   +14.475, E3 +78065.291}
SPL {X  -159.796, Y  +383.921, Z    +0.000, E1   +14.466, E3 +78085.947}
SPL {X  -159.651, Y  +381.443, Z    +0.000, E1   +14.453, E3 +78106.495}
SPL {X  -159.474, Y  +379.042, Z    +0.000, E1   +14.434, E3 +78126.459}
SPL {X  -159.316, Y  +377.219, Z    +0.000, E1   +14.400, E3 +78141.687}
ENDSPLINE

